(* CODESYS project 1_2_3_plc_chalet_xplanar.library
   Title: CHALET_XPlanar
   Version: 1.2.3
   Placeholder: CHALET_XPlanar
   Company: Beckhoff CH

Project tree, tasks and I/O mapping:
  libraries: CHALET_BaseComponents, * (Beckhoff CH); Tc2_Math, * (Beckhoff Automation GmbH); Tc2_Standard, 3.3.3.0 (Beckhoff Automation GmbH); Tc2_System, 3.4.25.0 (Beckhoff Automation GmbH); Tc2_Utilities, 3.3.52.0 (Beckhoff Automation GmbH); Tc3_EventLogger, 3.1.30.0 (Beckhoff Automation GmbH); Tc3_JsonXml, 3.3.18.0 (Beckhoff Automation GmbH); Tc3_Mc3PlanarMotion, 3.1.10.11 (Beckhoff Automation GmbH); Tc3_Module, 3.3.21.0 (Beckhoff Automation GmbH); Tc3_Physics, 3.1.10.3 (Beckhoff Automation GmbH); Tc3_XPlanarUtility, 3.1.2203.3 (Beckhoff Automation GmbH & Co. KG)
  COMPONENTs/
    Casting/
      function ToMover [ST]
      function ToMoverPair [ST]
      function ToStation [ST]
      function ToTrack [ST]
    Environment/
      CD_XP_Environment
      function block FB_XP_Environment [ST]: AddToGroup, RemoveFromGroup, Clear, Configure, FB_init, HR, Initialize, OID, PlanarEnvironment, Update, UtilityEnvirement
      interface I_XP_Environment: AddToGroup, Clear, Configure, HR, Initialize, OID, PlanarEnvironment, RemoveFromGroup, Update, UtilityEnvirement
    Group/
      CD_XP_Groups
      function block FB_XP_Group [ST]: AddEnvironment, AddMover, AddTrack, Disable, Enable, FB_init, HR, Initialize, OID, Reset, Update
      interface I_XP_Group: AddEnvironment, AddMover, AddTrack, Disable, Enable, HR, Initialize, OID, Reset, Update
    Mover/
      Pair/
        function block FB_XP_MoverPair [ST]: FB_init, MoverMaster, MoverSlave
        interface I_XP_MoverPair: MoverMaster, MoverSlave
      Single/
        function block FB_XP_Mover [ST]: AddToGroup, RemoveFromGroup, MoveC, Disable, Enable, Reset, JoinTrack, MoveOnTrack, PositionOnTrack, CurrentStation, DistToTrack, FB_init, Halt, HR, Initialize, Mode, OID, PlanarMover, TargetStation, TcIoXPlanarMover, Update, UpdatePosition, UtilityMover
        interface I_XP_Mover: AddToGroup, RemoveFromGroup, MoveC, Disable, Enable, Reset, JoinTrack, MoveOnTrack, PositionOnTrack, CurrentStation, DistToTrack, Halt, HR, Mode, OID, PlanarMover, TargetStation, TcIoXPlanarMover
        interface I_XP_Mover_PLC: OID, PlanarMover, TcIoXPlanarMover, UtilityMover
      CD_XP_Movers
    Stationen/
      function block FB_XP_Station_Base [ST]: Configure, Configuring, PlcIfaceToMover, AccocietedTrack, AddMoverToQueue, AssignedMovers, CtsFreeMoverBuffer, DeleteMoversQueue, Feedback, InterfaceToMover, IsMoverInStation, PositionOnTrack, PositionXY, Ready, SearchPathToTarged, SendMoverToGroup, SendMoverToGroupExp, StationGroupID, Update
      function block FB_XP_Station_FBinit [ST]: Configuring, FB_init
      function block FB_XP_Station_JSON [ST]: Configuring, FB_init
      interface I_XP_Station: AccocietedTrack, AddMoverToQueue, AssignedMovers, Configure, Configuring, DeleteMoversQueue, PositionOnTrack, SearchPathToTarged, SendMoverToGroup, SendMoverToGroupExp, StationGroupID, Update
      interface I_XP_Station_PLC: AccocietedTrack, Feedback, IsMoverInStation, PlcIfaceToMover, PositionOnTrack, PositionXY, Ready, SendMoverToGroup, StationGroupID
      Klassendiagramm
      data type ST_PathFinder
    System/
      CD_XP_System
      CD_XP_System_Objects
      function block FB_XP_System [ST]: Disable, Disabled, Disabling, Enable, Enabled, Enabling, Station, ValidLUID, LinkEnvironment, LinkGroup, RegisterMover, RegisterMoverPair, RegisterStation, RegisterTrack, JoiningStation, JoiningTrack, Enviroment, Feedback, Initialize, Movers, Stations, Tracks, Update
      interface I_XP_System_PLC: Disable, Disabled, Enable, Enabled, Feedback, Initialize, Station, Update, ValidLUID
      interface I_XP_System_Registration: Enviroment, LinkEnvironment, LinkGroup, Movers, RegisterMover, RegisterMoverPair, RegisterStation, RegisterTrack, Stations, Tracks
    Track/
      CD_XP_Track
      function block FB_XP_Track_Base [ST]: AddToGroup, RemoveFromGroup, AddMover, CalcTrackPoints, Configure, Configuring, Disable, Enable, FB_init, HR, Length, OID, PlanarTrack, Reset, Update
      function block FB_XP_Track_JSON [ST]: ReadCenter, ReadDirection, ReadEnd, ReadStart, Configuring
      function block FB_XP_Track_TcCom [ST]: Configuring
      interface I_XP_Track: AddMover, AddToGroup, CalcTrackPoints, Configure, Configuring, Disable, Enable, HR, Length, OID, PlanarTrack, RemoveFromGroup, Reset
    Class Diagram_Iface
  00000000-0000-0000-0000-000000000000|Disclaimer Standard DE R1006.pdf
  Disclaimer Standard DE R1006.pdf
  global variables XPlanarParameterlist
*)

// COMPONENTs/Stationen/ST_PathFinder
TYPE ST_PathFinder :
STRUCT
	bTargetFound : BOOL; // Targed Station found on this path. No information about ready or not	
	nDistToTarget : INT;
	iFoundStation : I_CH_Object;
END_STRUCT
END_TYPE

// XPlanarParameterlist
{attribute 'qualified_only'}
VAR_GLOBAL CONSTANT 
	(*Minimum gap center to center on track *)
	F_MOVER_MINIMUM_GAP_ON_TRACK : LREAL := 200.0;

	(*Additional gap center to center on track *)
	F_MOVER_ADDITIONAL_GAP_ON_TRACK : LREAL := 60.0;
	
	(*Pathfinder max recursion search depth in stations*)
	N_MAX_SEARCH_DEPTH: INT := 5;
		
	(*Use the automatic deployment function to copy the .JSON files to the %TC_BOOTPRJPATH%OCFG at Activate configuration*)
	S_JSON_FOLDER_PATH_ON_TARGED : STRING := 'C:\TwinCAT\3.1\Boot\OCFG\';
	
	(*get an array of points of track in this size *)
	N_TRACE_POINTS : UINT := 30;
END_VAR

// COMPONENTs/Casting/ToMover
FUNCTION ToMover : BOOL
VAR_INPUT
	iChObject : I_CH_OBJECT;
	iXpMover : Reference to I_XP_Mover;
END_VAR

VAR
	iTmp : I_XP_Mover;
END_VAR

(* 
   1. Test if the interface exists
   2. Test if the object implements a "Object" interface 
   3. Write reference to interface in parameter
   4. Returne TRUE if succesfull
*)
IF iChObject <> 0 AND_THEN __QUERYINTERFACE(iChObject,iTmp) THEN
	iXpMover := iTmp;
	ToMover := TRUE;
END_IF

END_FUNCTION

// COMPONENTs/Mover/Single/I_XP_Mover
INTERFACE I_XP_Mover EXTENDS __SYSTEM.IQueryInterface

METHOD AddToGroup : HRESULT
VAR_INPUT
	iGroup : I_XP_Group;
END_VAR
END_METHOD

METHOD RemoveFromGroup : HRESULT
END_METHOD

METHOD MoveC : HRESULT
VAR_INPUT
	fPosition : LREAL;
END_VAR
END_METHOD

METHOD Disable : HRESULT
VAR_INPUT
END_VAR
END_METHOD

METHOD Enable : HRESULT
VAR_INPUT
END_VAR
END_METHOD

METHOD Reset : HRESULT
VAR_INPUT
END_VAR
END_METHOD

METHOD JoinTrack : HRESULT
VAR_INPUT
	iTrack : I_XP_Track;
END_VAR
END_METHOD

METHOD MoveOnTrack : HRESULT
VAR_INPUT
	iTrack : I_XP_Track;
	fPosition : LREAL;
END_VAR
END_METHOD

PROPERTY PositionOnTrack : Lreal
GET
END_GET
END_PROPERTY

{attribute 'monitoring':='call'}
PROPERTY CurrentStation : STRING
GET
END_GET
SET
END_SET
END_PROPERTY

METHOD DistToTrack : LREAL
VAR_INPUT
	iTrack : I_XP_Track;
END_VAR
END_METHOD

METHOD Halt : HRESULT
VAR_INPUT
END_VAR
END_METHOD

{attribute 'monitoring':='call'}
PROPERTY HR : HRESULT
GET
END_GET
END_PROPERTY

{attribute 'monitoring':='call'}
PROPERTY Mode : MC_PLANAR_MOVER_COMMAND_MODE
GET
END_GET
END_PROPERTY

{attribute 'monitoring':='call'}
PROPERTY OID : OTCID
GET
END_GET
END_PROPERTY

{attribute 'monitoring':='call'}
PROPERTY PlanarMover : REFERENCE TO MC_PlanarMover
GET
END_GET
END_PROPERTY

{attribute 'monitoring':='call'}
PROPERTY TargetStation : String
GET
END_GET
SET
END_SET
END_PROPERTY

PROPERTY TcIoXPlanarMover : Tc3_XPlanarUtility.I_TcIoXPlanarMover
GET
END_GET
END_PROPERTY

END_INTERFACE

// COMPONENTs/Group/I_XP_Group
INTERFACE I_XP_Group

METHOD AddEnvironment : HRESULT
VAR_INPUT
	refEnvironment : REFERENCE TO MC_PlanarEnvironment;
	refFeedback : REFERENCE TO MC_PlanarFeedback;
END_VAR
END_METHOD

METHOD AddMover : HRESULT
VAR_INPUT
	refMover : REFERENCE TO MC_PlanarMover;
	refFeedback : REFERENCE TO MC_PlanarFeedback;
END_VAR
END_METHOD

METHOD AddTrack : HRESULT
VAR_INPUT
	refTrack : REFERENCE TO MC_PlanarTrack;
	refFeedback : REFERENCE TO MC_PlanarFeedback;
END_VAR
END_METHOD

METHOD Disable : HRESULT
VAR_INPUT
END_VAR
END_METHOD

METHOD Enable : HRESULT
VAR_INPUT
END_VAR
END_METHOD

{attribute 'monitoring':='call'}
PROPERTY HR : HRESULT
GET
END_GET
END_PROPERTY

METHOD Initialize : HRESULT
VAR_INPUT
END_VAR
END_METHOD

{attribute 'monitoring':='call'}
PROPERTY OID : OTCID
GET
END_GET
END_PROPERTY

METHOD Reset : HRESULT
VAR_INPUT
END_VAR
END_METHOD

METHOD PUBLIC Update : HRESULT
VAR_INPUT
END_VAR
END_METHOD

END_INTERFACE

// COMPONENTs/Track/I_XP_Track
INTERFACE I_XP_Track

METHOD AddMover : HRESULT
VAR_INPUT
	refMover : REFERENCE TO MC_PlanarMover;
	refFeedback : REFERENCE TO MC_PlanarFeedback;
END_VAR
END_METHOD

METHOD AddToGroup : HRESULT
VAR_INPUT
	iGroup : I_XP_Group;
END_VAR
END_METHOD

METHOD CalcTrackPoints : HRESULT
VAR_INPUT
END_VAR
END_METHOD

METHOD Configure : HRESULT
VAR_INPUT
END_VAR
END_METHOD

METHOD Configuring : HRESULT
VAR_INPUT
END_VAR
END_METHOD

METHOD Disable : HRESULT
VAR_INPUT
END_VAR
END_METHOD

METHOD Enable : HRESULT
VAR_INPUT
END_VAR
END_METHOD

{attribute 'monitoring':='call'}
PROPERTY HR : HRESULT
GET
END_GET
END_PROPERTY

{attribute 'monitoring':='call'}
PROPERTY Length : LREAL
GET
END_GET
END_PROPERTY

{attribute 'monitoring':='call'}
PROPERTY OID : OTCID
GET
END_GET
END_PROPERTY

{attribute 'monitoring':='call'}
PROPERTY PlanarTrack : REFERENCE TO MC_PlanarTrack
GET
END_GET
END_PROPERTY

METHOD RemoveFromGroup : HRESULT
END_METHOD

METHOD Reset : HRESULT
VAR_INPUT
END_VAR
END_METHOD

END_INTERFACE

// COMPONENTs/Casting/ToMoverPair
FUNCTION ToMoverPair : BOOL
VAR_INPUT
	iChObject : I_CH_OBJECT;
	iXpMoverPair : Reference to I_XP_MoverPair;
END_VAR

VAR
	iTmp : I_XP_MoverPair;
END_VAR

(* 
   1. Test if the interface exists
   2. Test if the object implements a "Object" interface 
   3. Write reference to interface in parameter
   4. Returne TRUE if succesfull
*)
IF iChObject <> 0 AND_THEN __QUERYINTERFACE(iChObject,iTmp) THEN
	iXpMoverPair := iTmp;
	ToMoverPair := TRUE;
END_IF

END_FUNCTION

// COMPONENTs/Mover/Pair/I_XP_MoverPair
INTERFACE I_XP_MoverPair

{attribute 'monitoring':='call'}
PROPERTY MoverMaster : I_XP_Mover
GET
END_GET
SET
END_SET
END_PROPERTY

{attribute 'monitoring':='call'}
PROPERTY MoverSlave : I_XP_Mover
GET
END_GET
SET
END_SET
END_PROPERTY

END_INTERFACE

// COMPONENTs/Casting/ToStation
FUNCTION ToStation : BOOL
VAR_INPUT
	iChObject : I_CH_OBJECT;
	iXpStation : REFERENCE TO I_XP_Station;
END_VAR

VAR
	iTmp : I_XP_Station;
END_VAR

(* Register the Station
   1. Test if the interface exists
   2. Test if the object implements a "Object" interface 
*)
IF iChObject <> 0 AND_THEN __QUERYINTERFACE(iChObject,iTmp) THEN
	iXpStation := iTmp;
	ToStation := TRUE;
END_IF

END_FUNCTION

// COMPONENTs/Stationen/I_XP_Station
INTERFACE I_XP_Station EXTENDS __SYSTEM.IQueryInterface

{attribute 'monitoring':='call'}
PROPERTY AccocietedTrack : I_XP_Track
GET
END_GET
END_PROPERTY

METHOD AddMoverToQueue : HRESULT
VAR_INPUT
	iMover : I_CH_Object;
END_VAR
END_METHOD

PROPERTY AssignedMovers : I_CH_List
GET
END_GET
END_PROPERTY

METHOD Configure : HRESULT
END_METHOD

METHOD Configuring : HRESULT
END_METHOD

METHOD DeleteMoversQueue : HRESULT
VAR_INPUT
END_VAR
END_METHOD

PROPERTY PositionOnTrack : LREAL
GET
END_GET
END_PROPERTY

METHOD SearchPathToTarged : ST_PathFinder
VAR_INPUT
	sTargedStationGroupId	: STRING;
	nSearchDepth		: INT;
END_VAR
END_METHOD

METHOD SendMoverToGroup : I_CH_Feedback
VAR_INPUT 
	sTargedStationGroupID : STRING;
END_VAR
END_METHOD

METHOD SendMoverToGroupExp : HRESULT
VAR_INPUT
	sTargedStationGroupID : STRING;
	iMover : I_XP_Mover;
END_VAR
END_METHOD

{attribute 'monitoring':='call'}
PROPERTY StationGroupID : STRING
GET
END_GET
END_PROPERTY

METHOD Update : HRESULT
VAR_INPUT
END_VAR
END_METHOD

END_INTERFACE

// COMPONENTs/Casting/ToTrack
FUNCTION ToTrack : BOOL
VAR_INPUT
	iChObject : I_CH_OBJECT;
	iXpTrack : REFERENCE TO I_XP_Track;
END_VAR

VAR
	iTmp : I_XP_Track;
END_VAR

(* 
   1. Test if the interface exists
   2. Test if the object implements a "Object" interface 
   3. Write reference to interface in parameter
   4. Returne TRUE if succesfull
*)
IF iChObject <> 0 AND_THEN __QUERYINTERFACE(iChObject,iTmp) THEN
	iXpTrack := iTmp;
	ToTrack := TRUE;
END_IF

END_FUNCTION

// COMPONENTs/Environment/FB_XP_Environment
{attribute 'no_explicit_call' := '[FB_ImageSource] Do not call the body - Stick to OOP'}
FUNCTION_BLOCK FB_XP_Environment EXTENDS FB_CH_Object IMPLEMENTS I_XP_Environment
VAR
	fbEnvironment : MC_PlanarEnvironment;
	fbUtilityEnvirement : FB_TcIoXPlanarEnvironment;
	{attribute 'hide'}
	iXpSystem : I_XP_System_Registration;
	fbActiveCmd : MC_PlanarFeedback;

END_VAR

METHOD AddToGroup : HRESULT
VAR_INPUT
	iGroup : I_XP_Group;
END_VAR
IF NOT THIS^.fbActiveCmd.Busy AND NOT THIS^.fbActiveCmd.Busy THEN
	iGroup.AddEnvironment(THIS^.fbEnvironment, THIS^.fbActiveCmd);
	AddToGroup := S_OK;
ELSE
	AddToGroup := S_FALSE;
END_IF
END_METHOD

METHOD RemoveFromGroup : HRESULT
IF NOT THIS^.fbActiveCmd.Busy THEN
	THIS^.fbEnvironment.RemoveFromGroup(THIS^.fbActiveCmd);
	RemoveFromGroup := S_OK;
ELSE
	RemoveFromGroup := S_FALSE;
END_IF
END_METHOD

METHOD Clear : HRESULT
THIS^.fbEnvironment.Clear(commandFeedback:=THIS^.fbActiveCmd);
Clear := S_OK;
END_METHOD

METHOD Configure : HRESULT
// To be automatically read from the Utility Stator info
// 06.2022 is read automaticli if Envirement Init Parameter has a link to XPLANAR TcCom Object.

THIS^.fbEnvironment.CreateBoundary(commandFeedback:=THIS^.fbActiveCmd);
Configure := S_OK;
END_METHOD

METHOD FB_init : BOOL
VAR_INPUT
	bInitRetains : BOOL; // if TRUE, the retain variables are initialized (warm start / cold start)
	bInCopyCode : BOOL;  // if TRUE, the instance afterwards gets moved into the copy code (online change)
	oSystem : I_CH_Object;
END_VAR
(* Register to the Xplanar System
   1. Test if the interface exists
   2. Test if the object implements a "System for Mover" interface 
*)
IF oSystem <> 0 AND_THEN __QUERYINTERFACE(oSystem,THIS^.iXpSystem) THEN
	THIS^.iXpSystem.LinkEnvironment(THIS^);
END_IF
END_METHOD

{attribute 'monitoring':='call'}
PROPERTY HR : HRESULT
GET
IF THIS^.fbActiveCmd.Busy THEN
	HR := S_PENDING;
END_IF

IF THIS^.fbActiveCmd.Done THEN
	HR := S_OK;
END_IF

IF THIS^.fbActiveCmd.Error THEN
	HR := E_FAIL;
END_IF
END_GET
END_PROPERTY

METHOD Initialize : HRESULT
VAR_INST
	bInitDone :BOOL := FALSE;
END_VAR
IF NOT bInitDone THEN
	Initialize := S_PENDING;
	IF fbUtilityEnvirement.Init(bExecute := TRUE) THEN
		fbUtilityEnvirement.Init(bExecute := FALSE);
		bInitDone := TRUE;
	END_IF
ELSE	
	Initialize := S_OK;
END_IF
END_METHOD

{attribute 'monitoring':='call'}
PROPERTY OID : OTCID
GET
OID := THIS^.fbEnvironment.MCTOPLC_STD.EnvironmentOID;
END_GET
END_PROPERTY

{attribute 'monitoring':='call'}
PROPERTY PlanarEnvironment : REFERENCE TO MC_PlanarEnvironment
GET
PlanarEnvironment ref= THIS^.fbEnvironment;
END_GET
END_PROPERTY

METHOD PUBLIC Update : HRESULT
VAR_INPUT
END_VAR
THIS^.fbEnvironment.Update();
fbActiveCmd.Update();
END_METHOD

PROPERTY UtilityEnvirement : Tc3_XPlanarUtility.I_Environment
GET
UtilityEnvirement := fbUtilityEnvirement;
END_GET
END_PROPERTY

END_FUNCTION_BLOCK

// COMPONENTs/Environment/I_XP_Environment
INTERFACE I_XP_Environment

METHOD AddToGroup : HRESULT
VAR_INPUT
	iGroup : I_XP_Group;
END_VAR
END_METHOD

METHOD Clear : HRESULT
END_METHOD

METHOD Configure : HRESULT
VAR_INPUT
END_VAR
END_METHOD

{attribute 'monitoring':='call'}
PROPERTY HR : HRESULT
GET
END_GET
END_PROPERTY

METHOD Initialize : HRESULT
END_METHOD

{attribute 'monitoring':='call'}
PROPERTY OID : OTCID
GET
END_GET
END_PROPERTY

{attribute 'monitoring':='call'}
PROPERTY PlanarEnvironment : REFERENCE TO MC_PlanarEnvironment
GET
END_GET
END_PROPERTY

METHOD RemoveFromGroup : HRESULT
END_METHOD

METHOD PUBLIC Update : HRESULT
VAR_INPUT
END_VAR
END_METHOD

PROPERTY UtilityEnvirement : Tc3_XPlanarUtility.I_Environment
GET
END_GET
END_PROPERTY

END_INTERFACE

// COMPONENTs/System/I_XP_System_Registration
INTERFACE I_XP_System_Registration

PROPERTY Enviroment : I_XP_Environment
GET
END_GET
END_PROPERTY

METHOD LinkEnvironment : HRESULT
VAR_INPUT
	oEnvironment : I_CH_Object;
END_VAR
END_METHOD

METHOD LinkGroup : HRESULT
VAR_INPUT
	oGroup : I_CH_Object;
END_VAR
END_METHOD

PROPERTY Movers : I_CH_LIST
GET
END_GET
END_PROPERTY

METHOD RegisterMover : HRESULT
VAR_INPUT
	oMover : I_CH_Object;
END_VAR
END_METHOD

METHOD RegisterMoverPair : HRESULT
VAR_INPUT
	oMoverPair : I_CH_Object;
END_VAR
END_METHOD

METHOD RegisterStation : HRESULT
VAR_INPUT
	oStation : I_CH_Object;
END_VAR
END_METHOD

METHOD RegisterTrack : HRESULT
VAR_INPUT
	oTrack : I_CH_Object;
END_VAR
END_METHOD

PROPERTY Stations : I_CH_LIST
GET
END_GET
END_PROPERTY

PROPERTY Tracks : I_CH_LIST
GET
END_GET
END_PROPERTY

END_INTERFACE

// COMPONENTs/Group/FB_XP_Group
{attribute 'no_explicit_call' := '[FB_ImageSource] Do not call the body - Stick to OOP'}
FUNCTION_BLOCK FB_XP_Group EXTENDS FB_CH_Object IMPLEMENTS I_XP_Group
VAR
	fbGroup : MC_PlanarGroup;
	{attribute 'hide'}
	iXpSystem : I_XP_System_Registration;
	fbActiveCmd : MC_PlanarFeedback;
END_VAR

METHOD AddEnvironment : HRESULT
VAR_INPUT
	refEnvironment : REFERENCE TO MC_PlanarEnvironment;
	refFeedback : REFERENCE TO MC_PlanarFeedback;
END_VAR
refEnvironment.AddToGroup(refFeedback, fbGroup);
END_METHOD

METHOD AddMover : HRESULT
VAR_INPUT
	refMover : REFERENCE TO MC_PlanarMover;
	refFeedback : REFERENCE TO MC_PlanarFeedback;
END_VAR
refMover.AddToGroup(refFeedback, fbGroup);
END_METHOD

METHOD AddTrack : HRESULT
VAR_INPUT
	refTrack : REFERENCE TO MC_PlanarTrack;
	refFeedback : REFERENCE TO MC_PlanarFeedback;
END_VAR
refTrack.AddToGroup(refFeedback, fbGroup);
END_METHOD

METHOD Disable : HRESULT
VAR_INPUT
END_VAR
IF NOT THIS^.fbActiveCmd.Busy THEN
	THIS^.fbGroup.Disable(fbActiveCmd);
	Disable := S_OK;
ELSE
	Disable := S_FALSE;
END_IF
END_METHOD

METHOD Enable : HRESULT
VAR_INPUT
END_VAR
IF NOT THIS^.fbActiveCmd.Busy THEN
	THIS^.fbGroup.Enable(fbActiveCmd);
	Enable := S_OK;
ELSE
	Enable := S_FALSE;
END_IF
END_METHOD

METHOD FB_init : BOOL
VAR_INPUT
	bInitRetains : BOOL; // if TRUE, the retain variables are initialized (warm start / cold start)
	bInCopyCode : BOOL;  // if TRUE, the instance afterwards gets moved into the copy code (online change)
	oSystem : I_CH_Object;
END_VAR
(* Register to the Xplanar System
   1. Test if the interface exists
   2. Test if the object implements a "System for Mover" interface 
*)
IF oSystem <> 0 AND_THEN __QUERYINTERFACE(oSystem,THIS^.iXpSystem) THEN
	THIS^.iXpSystem.LinkGroup(THIS^);
END_IF
END_METHOD

{attribute 'monitoring':='call'}
PROPERTY HR : HRESULT
GET
IF THIS^.fbActiveCmd.Busy THEN
	HR := S_PENDING;
END_IF

IF THIS^.fbActiveCmd.Done THEN
	HR := S_OK;
END_IF

IF THIS^.fbActiveCmd.Error THEN
	HR := E_FAIL;
END_IF
END_GET
END_PROPERTY

METHOD Initialize : HRESULT
VAR_INPUT
END_VAR
Initialize := S_OK;
END_METHOD

{attribute 'monitoring':='call'}
PROPERTY OID : OTCID
GET
OID := THIS^.fbGroup.MCTOPLC_STD.GroupOID;
END_GET
END_PROPERTY

METHOD Reset : HRESULT
VAR_INPUT
END_VAR
IF NOT THIS^.fbActiveCmd.Busy THEN
	THIS^.fbGroup.Reset(fbActiveCmd);
	Reset := S_OK;
ELSE
	Reset := S_FALSE;
END_IF
END_METHOD

METHOD PUBLIC Update : HRESULT
VAR_INPUT
END_VAR
THIS^.fbGroup.Update();
fbActiveCmd.Update();
END_METHOD

END_FUNCTION_BLOCK

// COMPONENTs/Mover/Pair/FB_XP_MoverPair
FUNCTION_BLOCK FB_XP_MoverPair EXTENDS FB_CH_Object IMPLEMENTS I_XP_MoverPair
VAR
	{attribute 'hide'}
    iMoverMaster : I_XP_Mover;
	{attribute 'hide'}
    iMoverSlave  : I_XP_Mover;
	{attribute 'hide'}
    iXpSystem    : I_XP_System_Registration;
END_VAR

METHOD FB_init : BOOL
VAR_INPUT
	bInitRetains : BOOL; // if TRUE, the retain variables are initialized (warm start / cold start)
	bInCopyCode : BOOL;  // if TRUE, the instance afterwards gets moved into the copy code (online change)
	oSystem : I_CH_Object;
END_VAR

VAR
	iXpSystem : I_XP_System_Registration;
END_VAR
(* Register to the Xplanar System
   1. Test if the interface exists
   2. Test if the object implements a "System for Mover" interface 
*)
IF oSystem <> 0 AND_THEN __QUERYINTERFACE(oSystem,THIS^.iXpSystem) THEN
	THIS^.iXpSystem.RegisterMoverPair(THIS^);
END_IF
END_METHOD

{attribute 'monitoring':='call'}
PROPERTY MoverMaster : I_XP_Mover
GET
MoverMaster := THIS^.iMoverMaster;
END_GET
SET
THIS^.iMoverMaster := MoverMaster;
END_SET
END_PROPERTY

{attribute 'monitoring':='call'}
PROPERTY MoverSlave : I_XP_Mover
GET
MoverSlave := THIS^.iMoverSlave;
END_GET
SET
THIS^.iMoverSlave := MoverSlave;
END_SET
END_PROPERTY

END_FUNCTION_BLOCK

// COMPONENTs/Mover/Single/FB_XP_Mover
// The warning " Interface of overridden methode xxx of base I_xxx doesn't match declaration" can be disabled here. 
{warning disable C0094 }

FUNCTION_BLOCK FB_XP_Mover EXTENDS FB_CH_Object IMPLEMENTS I_XP_Mover, I_XP_Mover_PLC
VAR
	fbMover : MC_PlanarMover;
	fbActiveCmd : MC_PlanarFeedback;	
	
	{attribute 'hide'} 
	fbUtilityMover : FB_McPlanarMover;
	{attribute 'hide'}
	iXpSystem : I_XP_System_Registration;
	{attribute 'hide'} 
	stPosition : PositionXYC;
	{attribute 'hide'} 
	sTargedStation : STRING;
	{attribute 'hide'} 
	sCurrentStation : STRING;
END_VAR

{warning restore C0094}

METHOD AddToGroup : HRESULT
VAR_INPUT
	iGroup : I_XP_Group;
END_VAR
IF NOT THIS^.fbActiveCmd.Busy THEN
	iGroup.AddMover(THIS^.fbMover, THIS^.fbActiveCmd);
	AddToGroup := S_OK;
ELSE
	AddToGroup := S_FALSE;
END_IF
END_METHOD

METHOD RemoveFromGroup : HRESULT

VAR
	iGroup: INT;
END_VAR
IF NOT THIS^.fbActiveCmd.Busy THEN
	THIS^.fbMover.RemoveFromGroup(THIS^.fbActiveCmd);
	RemoveFromGroup := S_OK;
ELSE
	RemoveFromGroup := S_FALSE;
END_IF
END_METHOD

METHOD MoveC : HRESULT
VAR_INPUT
	fPosition : LREAL;
END_VAR

THIS^.fbMover.MoveC(commandFeedback	:= THIS^.fbActiveCmd, 
					targetPosition	:= fPosition, 
					constraint		:= 0, 
					options			:= 0
					);

MoveC := S_OK;
END_METHOD

METHOD Disable : HRESULT
VAR_INPUT
END_VAR
THIS^.fbMover.Disable(THIS^.fbActiveCmd);
Disable := S_OK;
END_METHOD

METHOD Enable : HRESULT
VAR_INPUT
END_VAR
IF NOT THIS^.fbActiveCmd.Busy THEN
	THIS^.fbMover.Enable(fbActiveCmd);
	Enable := S_OK;
ELSE
	Enable := S_FALSE;
END_IF
END_METHOD

METHOD Reset : HRESULT
VAR_INPUT
END_VAR
THIS^.fbMover.Reset(THIS^.fbActiveCmd);
Reset := S_OK;
END_METHOD

METHOD JoinTrack : HRESULT
VAR_INPUT
	iTrack : I_XP_Track;
END_VAR

VAR
	//iTrack : I_XP_Track;
END_VAR
IF NOT THIS^.fbActiveCmd.Busy THEN
	iTrack.AddMover(THIS^.fbMover, THIS^.fbActiveCmd);
	JoinTrack := S_OK;
ELSE
	JoinTrack := S_FALSE;
END_IF
END_METHOD

METHOD MoveOnTrack : HRESULT
VAR_INPUT
	iTrack : I_XP_Track;
	fPosition : LREAL;
END_VAR

VAR
	moveOptions: ST_MoveOnTrackOptions;
	fMoverDiagonal : LREAL;
END_VAR
moveOptions.direction := MC_DIRECTION.mcDirectionPositive;
moveOptions.additionalTurns := 0;

//gap = Pythagoras diagonal + x mm, minimum x mm
fMoverDiagonal := SQRT(EXPT((THIS^.fbUtilityMover.GetMoverHeight()),2)+EXPT((THIS^.fbUtilityMover.GetMoverWidth()),2));
moveOptions.gap := MAX(XPlanarParameterlist.F_MOVER_MINIMUM_GAP_ON_TRACK ,fMoverDiagonal + XPlanarParameterlist.F_MOVER_ADDITIONAL_GAP_ON_TRACK );

IF iTrack <> 0 THEN
	THIS^.fbMover.MoveOnTrack(
		commandFeedback:=THIS^.fbActiveCmd,
		targetTrack:=iTrack.PlanarTrack, 
		targetPositionOnTrack:=fPosition, 
		constraint:=0, 
		options:=moveOptions);
	MoveOnTrack := S_OK;
ELSE
	MoveOnTrack := S_FALSE;
END_IF
END_METHOD

PROPERTY PositionOnTrack : LREAL
GET
VAR
	fbMoverSetPosOnTrack: Tc3_XPlanarUtility.ST_MCMoverSetPosOnTrack;
END_VAR
fbMoverSetPosOnTrack := THIS^.fbUtilityMover.GetPositionOnTrack();
PositionOnTrack := fbMoverSetPosOnTrack.SetPos;
END_GET
END_PROPERTY

{attribute 'monitoring':='call'}
PROPERTY CurrentStation : STRING
GET
CurrentStation := THIS^.sCurrentStation;
END_GET
SET
THIS^.sCurrentStation := currentStation;
END_SET
END_PROPERTY

METHOD DistToTrack : LREAL
VAR_INPUT
	iTrack : I_XP_Track;
END_VAR
VAR
	fPositionOnTrack : LREAL;
	trackPosition : PositionXYC;
END_VAR
//get Pos on track in mm
fPositionOnTrack := iTrack.PlanarTrack.GetArcLengthClosestTo(geometry:=THIS^.stPosition);

//convert pos on track in XY
iTrack.PlanarTrack.GetPositionAt(arcLength := fPositionOnTrack, position:=trackPosition);

//get distance to mover
DistToTrack := SQRT(EXPT((trackPosition.x - THIS^.stPosition.x),2)+EXPT((trackPosition.y - THIS^.stPosition.y),2));
END_METHOD

METHOD FB_init : BOOL
VAR_INPUT
	bInitRetains : BOOL; // if TRUE, the retain variables are initialized (warm start / cold start)
	bInCopyCode : BOOL;  // if TRUE, the instance afterwards gets moved into the copy code (online change)
	oSystem : I_CH_Object;
END_VAR
(* Register to the Xplanar System
   1. Test if the interface exists
   2. Test if the object implements a "System for Mover" interface 
*)
IF oSystem <> 0 AND_THEN __QUERYINTERFACE(oSystem,THIS^.iXpSystem) THEN
	THIS^.iXpSystem.RegisterMover(THIS^);
END_IF
END_METHOD

METHOD Halt : HRESULT
VAR_INPUT
END_VAR
THIS^.fbMover.Halt(THIS^.fbActiveCmd,0);

Halt := S_OK;
END_METHOD

{attribute 'monitoring':='call'}
PROPERTY HR : HRESULT
GET
IF THIS^.fbActiveCmd.Busy THEN 
	HR := S_PENDING;
END_IF

IF THIS^.fbActiveCmd.Done THEN 
	HR := S_OK;
END_IF

IF THIS^.fbActiveCmd.Error THEN 
	HR := E_FAIL;
END_IF
END_GET
END_PROPERTY

METHOD Initialize : HRESULT
VAR_INST
	bInitDone :BOOL := FALSE;
END_VAR
VAR
	//nLoopIndex : UINT;
	
	//zzzMover : I_TcIoXPlanarMover;
	//zzzTcIoXPlanar : I_TcIoXPlanarProcessingUnit;
	//zzzOid : OTCID;
	//zzzIENv : I_XP_Environment;
END_VAR
IF NOT bInitDone THEN
	Initialize := S_PENDING;
	
	//braucht es das noch? zzz
	//IF iXpSystem.Enviroment.Initialize() <> S_OK  THEN
	//	//wait until init of FB_TcIoXPlanarEnvironment is done.
	//	RETURN;
	//END_IF
	//
    //
	//IF fbUtilityMover.Init(bExecute:= TRUE, nObjectId:=THIS^.fbMover.MCTOPLC.STD.MoverOID) THEN
	//	fbUtilityMover.Init(bExecute:= FALSE, nObjectId:=THIS^.fbMover.MCTOPLC.STD.MoverOID);
	//ELSE
	//	RETURN;
	//END_IF
		
	bInitDone := TRUE;	
	
ELSE	
	Initialize := S_OK;	
END_IF
END_METHOD

{attribute 'monitoring':='call'}
PROPERTY Mode : MC_PLANAR_MOVER_COMMAND_MODE
GET
Mode := THIS^.fbMover.MCTOPLC.STD.CommandMode;
END_GET
END_PROPERTY

{attribute 'monitoring':='call'}
PROPERTY OID : OTCID
GET
OID := THIS^.fbMover.MCTOPLC.STD.MoverOID;
END_GET
END_PROPERTY

{attribute 'monitoring':='call'}
PROPERTY PlanarMover : REFERENCE TO MC_PlanarMover
GET
PlanarMover ref= THIS^.fbMover;
END_GET
END_PROPERTY

{attribute 'monitoring':='call'}
PROPERTY TargetStation : String
GET
TargetStation := THIS^.sTargedStation;
END_GET
SET
THIS^.sTargedStation := TargetStation;
END_SET
END_PROPERTY

{attribute 'monitoring':='call'}
PROPERTY TcIoXPlanarMover : Tc3_XPlanarUtility.I_TcIoXPlanarMover
GET
VAR
	nLoopIndex : UINT;
	zzzMover : I_TcIoXPlanarMover;
END_VAR
//TcIoXPlanarMover:= THIS^.iTcIoXPlanarMover;

FOR nLoopIndex := 1 TO UDINT_TO_UINT(Param_TcIoXPlanarEnvironment.MaxXPlanarMoversPerXpu) DO
	zzzMover := iXpSystem.Enviroment.UtilityEnvirement.XpuTcIo(1).MoverTcIo(nLoopIndex);
	IF zzzMover <> 0 AND_THEN zzzMover.GetNcMoverOid() = OID THEN
		TcIoXPlanarMover := iXpSystem.enviroment.UtilityEnvirement.XpuTcIo(1).MoverTcIo(nLoopIndex);
		RETURN;
	END_IF
END_FOR
END_GET
END_PROPERTY

METHOD PUBLIC Update : HRESULT
VAR_INPUT
END_VAR
THIS^.fbMover.Update();
THIS^.fbActiveCmd.Update();

THIS^.UpdatePosition();
END_METHOD

METHOD UpdatePosition : HRESULT
VAR_INPUT
END_VAR
THIS^.stPosition.x := THIS^.fbMover.MCTOPLC.ACT.ActPos.x;
THIS^.stPosition.y := THIS^.fbMover.MCTOPLC.ACT.ActPos.y;
THIS^.stPosition.c := THIS^.fbMover.MCTOPLC.ACT.ActPos.c;
END_METHOD

{attribute 'monitoring':='call'}
PROPERTY UtilityMover : I_McPlanarMover
GET
UtilityMover := THIS^.fbUtilityMover;
END_GET
END_PROPERTY

END_FUNCTION_BLOCK

// COMPONENTs/Mover/Single/I_XP_Mover_PLC
INTERFACE I_XP_Mover_PLC

{attribute 'monitoring':='call'}
PROPERTY OID : OTCID
GET
END_GET
END_PROPERTY

{attribute 'monitoring':='call'}
PROPERTY PlanarMover : REFERENCE TO MC_PlanarMover
GET
END_GET
END_PROPERTY

PROPERTY TcIoXPlanarMover : Tc3_XPlanarUtility.I_TcIoXPlanarMover
GET
END_GET
END_PROPERTY

{attribute 'monitoring':='call'}
PROPERTY UtilityMover : I_McPlanarMover
GET
END_GET
END_PROPERTY

END_INTERFACE

// COMPONENTs/Stationen/FB_XP_Station_Base
FUNCTION_BLOCK ABSTRACT FB_XP_Station_Base EXTENDS FB_CH_Object IMPLEMENTS I_XP_Station, I_XP_Station_PLC
VAR
	{attribute 'hide'}
	bReady 		: BOOL := TRUE;
	{attribute 'hide'}
	sStationGroupID : STRING;
	{attribute 'hide'}
	nCtsMinMovers : INT := 0;
	{attribute 'hide'}
	nCtsMaxMovers : INT := 1;
	{attribute 'hide'}	
	fbPosition : PositionXY;
	{attribute 'hide'}	
	fbJsonParser : FB_JsonDomParser;
	{attribute 'hide'}	
	nState_Configuring: INT;
	{attribute 'hide'}	
	iAccocietedTrack : I_XP_Track;
	{attribute 'hide'}	
	iXpSystem : I_XP_System_Registration;
	
	{attribute 'hide'}
	fbFeedback : FB_CH_Feedback;
	
	(*List of stations*)
	{attribute 'hide'}	
	fbStationsAhead : FB_CH_List;
	
	(* Lists to handle the ownership of movers *)
	{attribute 'hide'}
	fbAssignedMovers 			: FB_CH_List;		// Movers approaching the station

END_VAR

METHOD Configure : HRESULT
VAR_INPUT
END_VAR
THIS^.nState_Configuring := 10;

Configure := S_OK;
END_METHOD

METHOD Abstract Configuring : HRESULT
VAR_INPUT
END_VAR
END_METHOD

{attribute 'monitoring':='call'}
(* Return interface to mover in station. Return 0 if no mover is in station *)
PROPERTY PlcIfaceToMover : I_XP_Mover_PLC
GET
VAR
	iMover : I_XP_Mover;
END_VAR
iMover := THIS^.InterfaceToMover;

IF 	iMover <> 0 THEN
	__QUERYINTERFACE(iMover,PlcIfaceToMover);
END_IF
END_GET
END_PROPERTY

{attribute 'monitoring':='call'}
PROPERTY AccocietedTrack : I_XP_Track
GET
AccocietedTrack := THIS^.iAccocietedTrack;
END_GET
END_PROPERTY

METHOD AddMoverToQueue : HRESULT
VAR_INPUT
	iMover : I_CH_Object;
END_VAR
VAR 
	iXPMover : I_XP_Mover;
END_VAR
IF ToMover(iMover, iXpMover) THEN
	AddMoverToQueue := fbAssignedMovers.AddObject(iMover);
	iXpMover.CurrentStation := THIS^.sStationGroupID;
ELSE
	AddMoverToQueue := E_FAIL;
END_IF
END_METHOD

PROPERTY AssignedMovers : I_CH_List
GET
AssignedMovers := THIS^.fbAssignedMovers;
END_GET
END_PROPERTY

//Return the number of avaiable moverplaces in this station. Return -1 if Station is not ready
{attribute 'monitoring':='call'}
PROPERTY CtsFreeMoverBuffer : INT
GET
VAR
	nMoversTotal: UINT;
END_VAR
IF NOT bReady THEN
	CtsFreeMoverBuffer := -1;
	RETURN;
END_IF

nMoversTotal := THIS^.fbAssignedMovers.Size;
CtsFreeMoverBuffer := THIS^.nCtsMaxMovers - TO_INT(nMoversTotal);
END_GET
END_PROPERTY

METHOD DeleteMoversQueue : HRESULT
VAR_INPUT
END_VAR
fbAssignedMovers.Clear();

DeleteMoversQueue := S_OK;
END_METHOD

{attribute 'monitoring':='call'}
PROPERTY Feedback : I_CH_Feedback
GET
Feedback := THIS^.fbFeedback;
END_GET
END_PROPERTY

{attribute 'monitoring':='call'}
(* Return interface to mover in station. Return 0 if no mover is in station *)
PROPERTY InterfaceToMover : I_XP_Mover
GET
VAR
	oMover : I_CH_Object;
	iMover : I_XP_Mover;
END_VAR
VAR CONSTANT
	fToleranceMm : LREAL := 1.0; 
END_VAR
InterfaceToMover := 0;

//compare all movers in this station with the coordinats of the station
THIS^.fbAssignedMovers.ResetIterator();
WHILE THIS^.fbAssignedMovers.HasNextObject() DO
	oMover := THIS^.fbAssignedMovers.GetNextObject();
	IF ToMover(oMover,iMover) THEN
		IF iMover.TargetStation = THIS^.StationGroupID 
			AND (iMover.HR = S_OK) //No active move cmd= Pos reached
			//AND (ABS(iMover.PlanarMover.MCTOPLC.SET.SetPos.x -  THIS^.fbPosition.x)<=fToleranceMm) 
			//AND (ABS(iMover.PlanarMover.MCTOPLC.SET.SetPos.y -  THIS^.fbPosition.y)<=fToleranceMm) 
			THEN	
			InterfaceToMover := iMover;
			RETURN;
		END_IF
	END_IF
END_WHILE
END_GET
END_PROPERTY

//Return TRUE if an mover is exactly on the station coordinates and has this station as destination
{attribute 'monitoring':='call'}
PROPERTY IsMoverInStation : BOOL
GET
//If interface to first mover is valid
IsMoverInStation := THIS^.InterfaceToMover<>0;
END_GET
END_PROPERTY

PROPERTY PositionOnTrack : LREAL
GET
PositionOnTrack := THIS^.iAccocietedTrack.PlanarTrack.GetArcLengthClosestTo(geometry:= THIS^.fbPosition);
END_GET
END_PROPERTY

{attribute 'monitoring':='call'}
PROPERTY PositionXY : REFERENCE TO  PositionXY
GET
PositionXY REF= THIS^.fbPosition;
END_GET
END_PROPERTY

{attribute 'monitoring':='call'}
PROPERTY Ready : BOOL
GET
Ready := THIS^.bReady;
END_GET
SET
THIS^.bReady := Ready;
END_SET
END_PROPERTY

METHOD SearchPathToTarged : ST_PathFinder
VAR_INPUT
	sTargedStationGroupId	: STRING;
	nSearchDepth			: INT;
END_VAR

VAR
	iStation: I_XP_Station;
	tempPath : ST_PathFinder;
	bestPath : ST_PathFinder;
END_VAR
//This is the serched Station
IF THIS^.sStationGroupID = sTargedStationGroupId THEN
	searchPathToTarged.iFoundStation := (THIS^);
	searchPathToTarged.nDistToTarget := 0;
	searchPathToTarged.bTargetFound := TRUE;
	
	//Station is full/not ready and can not be used as next targed
	IF THIS^.CtsFreeMoverBuffer <= 0 THEN
		searchPathToTarged.iFoundStation := 0;
	END_IF
	RETURN;
END_IF	


//Abort
IF nSearchDepth = XPlanarParameterlist.N_MAX_SEARCH_DEPTH THEN
	searchPathToTarged.iFoundStation := 0;
	searchPathToTarged.nDistToTarget := 0;
	searchPathToTarged.bTargetFound := FALSE;
END_IF


//seach on all station ahead the shortest way to targed
bestPath.nDistToTarget := 32767;
THIS^.fbStationsAhead.ResetIterator();
WHILE THIS^.fbStationsAhead.HasNextObject() DO
	IF ToStation(THIS^.fbStationsAhead.GetNextObject(),iStation) THEN
		tempPath := iStation.searchPathToTarged(sTargedStationGroupId, nSearchDepth+1);
		tempPath.nDistToTarget := tempPath.nDistToTarget +1;		
		IF tempPath.bTargetFound AND ((tempPath.nDistToTarget <= bestPath.nDistToTarget AND tempPath.iFoundStation<>0) OR (tempPath.nDistToTarget <= bestPath.nDistToTarget AND bestPath.iFoundStation=0)) THEN
			bestPath := tempPath;
		END_IF
	END_IF
END_WHILE


//Only check if the station is empty to pass through, if the station is not where the mover starts(the mover is there at first position)
IF nSearchDepth <> 0 THEN
	//IF current station has object, its not posible to move direct to next station, in this case use this station as targed
	IF bestPath.bTargetFound AND (NOT THIS^.fbAssignedMovers.IsEmpty OR bestPath.iFoundStation = 0)THEN
		//If the currend station has some empty buffer, use this as targed, else clear target and try in station before again
		IF THIS^.CtsFreeMoverBuffer > 0 THEN
			bestPath.iFoundStation := (THIS^);
		ELSE
			bestPath.iFoundStation := 0; 
		END_IF
	END_IF
END_IF


searchPathToTarged := bestPath;
END_METHOD

METHOD SendMoverToGroup : I_CH_Feedback
VAR_INPUT 
	sTargedStationGroupID : STRING;
END_VAR
VAR
	iMover : I_XP_Mover;
	sCommand : STRING;
END_VAR
IF THIS^.fbFeedback.Error THEN
	//Error active/not ready
	THIS^.fbFeedback.LastCommandAccepted	:= FALSE;

ELSIF NOT THIS^.IsMoverInStation THEN
	//No Mover in Station
	THIS^.fbFeedback.LastCommandAccepted	:= FALSE;

ELSIF sTargedStationGroupID=''  THEN
	//No targed
	THIS^.fbFeedback.LastCommandAccepted	:= FALSE;
	
ELSE
	iMover := THIS^.InterfaceToMover;
	//search path and send away.
	THIS^.fbFeedback.HR := THIS^.sendMoverToGroupExp(sTargedStationGroupID:=sTargedStationGroupID, iMover);
	
	//build string with command
	sCommand := CONCAT(sCommand,'sendMover');
	sCommand := CONCAT(sCommand, UDINT_TO_STRING(iMover.OID));
	sCommand := CONCAT(sCommand,'ToGroup');
	sCommand := CONCAT(sCommand,sTargedStationGroupID);	
	
	//set fbFeedback
	THIS^.fbFeedback.ActiveCommand		 := sCommand;
	THIS^.fbFeedback.LastCommandAccepted := TRUE;
END_IF

sendMoverToGroup := THIS^.fbFeedback;
END_METHOD

METHOD SendMoverToGroupExp : HRESULT
VAR_INPUT
	sTargedStationGroupID : STRING;
	iMover : I_XP_Mover;
END_VAR

VAR
	iMoverObject : I_CH_Object;
	iStation: I_XP_Station;
	pathForMover: ST_PathFinder;
END_VAR
IF iMover <> 0 THEN
	
	//set targed
	iMover.TargetStation := sTargedStationGroupID;
	
	//get object
	iMoverObject := THIS^.iXpSystem.Movers.FindOID(iMover.OID);
	
	//init
	iStation := THIS^;
	
	//remove mover from station(the search path metohde maybe not found an solution if this station is already full.
	THIS^.fbAssignedMovers.RemoveObject(iMoverObject);
	
	//search best station
	pathForMover := THIS^.searchPathToTarged(sTargedStationGroupId:= iMover.TargetStation, nSearchDepth:=0);

	IF NOT pathForMover.bTargetFound THEN
		// no path found in maximum search depth - ERROR
		sendMoverToGroupExp := E_FAIL;
	ELSIF pathForMover.iFoundStation = 0 THEN
		// path found but no movement posible, next station is full
		sendMoverToGroupExp := S_FALSE;
	ELSIF ToStation(pathForMover.iFoundStation,iStation) THEN
		//path found. valide interface. move to station
		sendMoverToGroupExp := iMover.MoveOnTrack(iTrack:=iStation.AccocietedTrack, fPosition:= iStation.PositionOnTrack);
	END_IF
	
	//Add mover to current or found station
	iStation.AddMoverToQueue(iMoverObject);

ELSE
	//Input not valide - ERROR
	SendMoverToGroupExp := E_FAIL;
END_IF
END_METHOD

{attribute 'monitoring':='call'}
PROPERTY StationGroupID : STRING
GET
StationGroupID := THIS^.sStationGroupId;
END_GET
END_PROPERTY

METHOD Update : HRESULT
VAR
	oMover: I_CH_Object;
	iMover: I_XP_MOVER;
	iStation: I_XP_Station;
	pathForFirstMoverInQue: ST_PathFinder;
END_VAR
VAR CONSTANT
	fToleranceMm : LREAL := 1.0; 
END_VAR
//get the first mover in the station queue(the mover at station coordinates)
//all movers are checked here, even those that do not have this station as a destination. Possibly the movers wait in this station until the next station becomes free.
THIS^.fbAssignedMovers.ResetIterator();
WHILE THIS^.fbAssignedMovers.HasNextObject() DO
	IF ToMover(THIS^.fbAssignedMovers.GetNextObject(),iMover) AND_THEN (iMover.HR = S_OK) THEN
			 //Found an mover in this station! Done= Targed reached, PEnding= Moving or an mover in the way
			 // check if first mover has another target than this station. Send away to targed
				IF iMover.TargetStation <> THIS^.StationGroupID AND iMover.TargetStation <> '' THEN
					THIS^.sendMoverToGroupExp(iMover:=iMover, sTargedStationGroupID:= iMover.TargetStation);
				END_IF			 
			 //Exit WHILE Loop
			EXIT;
	END_IF
END_WHILE


Update := S_OK;
END_METHOD

END_FUNCTION_BLOCK

// COMPONENTs/Stationen/I_XP_Station_PLC
INTERFACE I_XP_Station_PLC

{attribute 'monitoring':='call'}
PROPERTY AccocietedTrack : I_XP_Track
GET
END_GET
END_PROPERTY

{attribute 'monitoring':='call'}
PROPERTY Feedback : I_CH_Feedback
GET
END_GET
END_PROPERTY

//Return TRUE if an mover is exactly on the station coordinates and has this station as destination
{attribute 'monitoring':='call'}
PROPERTY IsMoverInStation : BOOL
GET
END_GET
END_PROPERTY

{attribute 'monitoring':='call'}
(* Return interface to mover in station. Return 0 if no mover is in station *)
PROPERTY PlcIfaceToMover : I_XP_Mover_PLC
GET
END_GET
END_PROPERTY

PROPERTY PositionOnTrack : LREAL
GET
END_GET
END_PROPERTY

{attribute 'monitoring':='call'}
PROPERTY PositionXY : REFERENCE TO  PositionXY
GET
END_GET
END_PROPERTY

{attribute 'monitoring':='call'}
PROPERTY Ready : BOOL
GET
END_GET
SET
END_SET
END_PROPERTY

METHOD SendMoverToGroup : I_CH_Feedback
VAR_INPUT 
	sTargedStationGroupID : STRING;
END_VAR
END_METHOD

{attribute 'monitoring':='call'}
PROPERTY StationGroupID : STRING
GET
END_GET
END_PROPERTY

END_INTERFACE

// COMPONENTs/Stationen/FB_XP_Station_FBinit
// The warning " Interface of overridden methode xxx of base I_xxx doesn't match declaration" can be disabled here. 
{warning disable C0094 }
{attribute 'no_explicit_call' := '[FB_ImageSource] Do not call the body - Stick to OOP'}
FUNCTION_BLOCK FB_XP_Station_FBinit EXTENDS FB_XP_Station_Base


{warning restore C0094}

METHOD Configuring : HRESULT
VAR_INPUT
END_VAR
VAR

	fPosOnTrack : LREAL;
	tempPosition : PositionXYC;

END_VAR
Configuring := S_PENDING;
CASE nState_Configuring OF
	0: // Idle
		Configuring := S_OK;
		
	10:	//convert Station position to an valid position on track
		fPosOnTrack := THIS^.iAccocietedTrack.PlanarTrack.GetArcLengthClosestTo(geometry:= THIS^.fbPosition);
		THIS^.iAccocietedTrack.PlanarTrack.GetPositionAt(arcLength:= fPosOnTrack, position:=tempPosition);
		THIS^.fbPosition.SetValuesXY(tempPosition.x, tempPosition.y);
		

		nState_Configuring := 100;


		
   100: // Done
		Configuring := S_OK;
		nState_Configuring := 0;
		
END_CASE

IF fbJsonParser.ExceptionRaised() THEN
	Configuring := E_FAIL;
END_IF

///zzz TODO Errorhandling
END_METHOD

METHOD FB_init : BOOL
VAR_INPUT
	bInitRetains : BOOL; // if TRUE, the retain variables are initialized (warm start / cold start)
	bInCopyCode : BOOL;  // if TRUE, the instance afterwards gets moved into the copy code (online change)
	
	
	oSystem : I_CH_Object;
	
	
	iAccocietedTrack 	: I_XP_Track;//track on which the station is located
	sUniqueIdentification : STRING; //unique identification for this station
	sStationGroupID		: STRING;//to which group of stations does this station belong? e.g. several stations can belong to one 'Infeed' if this is implemented redundantly.
	nCtsMaxMovers 		: UINT;
	xPos, yPos			: LREAL;
	
	//what kind of stations can be reached from this station? several if it has a switch. otherwise it usually only has one
	aStationsAhead1 	: I_CH_Object;
	aStationsAhead2 	: I_CH_Object;
	aStationsAhead3 	: I_CH_Object;
END_VAR

VAR CONSTANT
	MAX_STATION_IN_FRONT : UINT := 3;
END_VAR

VAR 
	nIndex : UINT;
END_VAR
(* Register to the Xplanar System
   1. Test if the interface exists
   2. Test if the object implements a "System for Mover" interface 
*)
IF oSystem <> 0 AND_THEN __QUERYINTERFACE(oSystem,THIS^.iXpSystem) THEN
	THIS^.iXpSystem.RegisterStation(THIS^);
END_IF




THIS^.iAccocietedTrack 	:= iAccocietedTrack;
THIS^.fbSelf.sName		:= sUniqueIdentification;
THIS^.sStationGroupID 	:= sStationGroupID;
THIS^.nCtsMaxMovers 	:= UINT_TO_INT(nCtsMaxMovers);

THIS^.fbPosition.x := xPos;
THIS^.fbPosition.y := yPos;


THIS^.fbStationsAhead.AddObject(iChObject:=aStationsAhead1);
THIS^.fbStationsAhead.AddObject(iChObject:=aStationsAhead2);
THIS^.fbStationsAhead.AddObject(iChObject:=aStationsAhead3);
END_METHOD

END_FUNCTION_BLOCK

// COMPONENTs/Stationen/FB_XP_Station_JSON
// The warning " Interface of overridden methode xxx of base I_xxx doesn't match declaration" can be disabled here. 
{warning disable C0094 }
{attribute 'no_explicit_call' := '[FB_ImageSource] Do not call the body - Stick to OOP'}
FUNCTION_BLOCK FB_XP_Station_JSON  EXTENDS FB_XP_Station_Base
(*
VAR
	{attribute 'hide'}
	bReady 		: BOOL := TRUE;
	{attribute 'hide'}
	sStationGroupID : STRING;
	{attribute 'hide'}
	nCtsMinMovers : INT := 0;
	{attribute 'hide'}
	nCtsMaxMovers : INT := 1;
	{attribute 'hide'}	
	fbPosition : PositionXY;
	{attribute 'hide'}	
	fbJsonParser : FB_JsonDomParser;
	{attribute 'hide'}	
	nState_Configuring: INT;
	{attribute 'hide'}	
	iAccocietedTrack : I_XP_Track;
	{attribute 'hide'}	
	iXpSystem : I_XP_System_Registration;
	
	{attribute 'hide'}
	fbFeedback : FB_CH_Feedback;
	
	(*List of stations*)
	{attribute 'hide'}	
	fbStationsAhead : FB_CH_List;
	
	(* Lists to handle the ownership of movers *)
	{attribute 'hide'}
	fbAssignedMovers 			: FB_CH_List;		// Movers approaching the station

END_VAR
*)
{warning restore C0094}

METHOD Configuring : HRESULT
VAR_INPUT
END_VAR

VAR_INST
    oDocument    : SJsonValue;
	oListOfStations: SJsonValue;
	oListOfStationsAhead: SJsonValue;
	oThisStation : SJsonValue;
	
	
    bExec        : BOOL;

    sPathFull    : STRING;
	
	oItr      : SJsonValue;
    oItrEnd   : SJsonValue;
END_VAR

VAR
    sType      : STRING(10);
	fType 		:LREAL;
	
	iFoundObject : I_CH_Object;
	iTrack : I_XP_Track;

    oProperty : SJsonValue;

	fPosOnTrack : LREAL;
	tempPosition : PositionXYC;

	lrDistMm : LREAL;
END_VAR
Configuring := S_PENDING;
CASE nState_Configuring OF
	0: // Idle
		Configuring := S_OK;
		
	10: // Clear
		// Clear Unique Id
		THIS^.fbSelf.sName := '';
		// delete list of stations ahead
		THIS^.fbStationsAhead.Clear();	
		nState_Configuring := 15;

	15:	// Configure file and load it
		bExec := TRUE;
		sPathFull := XPlanarParameterlist.S_JSON_FOLDER_PATH_ON_TARGED;
		sPathFull := CONCAT(sPathFull,'XP_Stations');
		sPathFull := CONCAT(sPathFull,'.JSON');	
		nState_Configuring := 20;
		
	20: // Load file
		fbJsonParser.LoadDocumentFromFile(sPathFull, bExec);
		IF NOT bExec THEN
			nState_Configuring := 30;
		END_IF
		
	30:	// Loading file		
		oDocument := fbJsonParser.GetDocumentRoot();
		nState_Configuring := 40;
	
	40: // Check file assgnment, load list
		oListOfStations := fbJsonParser.FindMember(oDocument, 'Stations');
	  	IF (oListOfStations <> 0) THEN
		    oItr := fbJsonParser.ArrayBegin(oListOfStations);
		    oItrEnd := fbJsonParser.ArrayEnd(oListOfStations);
			
			nState_Configuring := 50;
		ELSE 
			;//wrong file
	  	END_IF


	50: // Load single segment. Check all station is the Unique ID is already in use, else set it in this station
		IF oItr <> 0 AND_THEN oItrEnd <> 0 AND_THEN oItr <> oItrEnd THEN
			(* Determine segment type *)
			oProperty := fbJsonParser.FindMember(oItr,'LUID');
			sType := fbJsonParser.GetString(oProperty);
			iFoundObject := iXpSystem.Stations.FindLUID(sLUID:=sType);
			IF iFoundObject = 0 THEN
				//not found = this station can use the LUID
				THIS^.fbSelf.sName := sType;
				oThisStation:= oItr;
				nState_Configuring := 70;
			ELSE
				//the LUID is already in use by an other station. try next
				oItr := fbJsonParser.NextArray(oItr);
				nState_Configuring := 50;
			END_IF
		ELSE
		; //End of list. to many stations in PLC
		END_IF	
		
	70: //Writte JSON to Object  -  AccocietedTrack
		oProperty := fbJsonParser.FindMember(oThisStation,'AccocietedTrack');
		sType := fbJsonParser.GetString(oProperty);
		iFoundObject := iXpSystem.Tracks.FindOIDString(sType);
		
		IF iFoundObject <> 0  AND_THEN ToTrack(iFoundObject, iTrack) THEN
			THIS^.iAccocietedTrack := iTrack;
			nState_Configuring := 72;
		ELSE
			;//Error, Track not found			
		END_IF
		
		
	72: //Writte JSON to Object  -  StationGroupId
		oProperty := fbJsonParser.FindMember(oThisStation,'StationGroupId');
		sType := fbJsonParser.GetString(oProperty);
		
		IF sType <> '' THEN
			THIS^.sStationGroupID := sType;
			nState_Configuring := 74;
		ELSE
			;//Error, StationGroupId not found			
		END_IF		
		
	74: //Writte JSON to Object  -  CtsMaxMovers
		oProperty := fbJsonParser.FindMember(oThisStation,'CtsMaxMovers');
		fType := fbJsonParser.GetDouble(oProperty);
		THIS^.nCtsMaxMovers := LREAL_TO_INT(fType);
		nState_Configuring := 76;
		
	76: //Writte JSON to Object  -  Position
		oProperty := fbJsonParser.FindMemberPath(oThisStation,'Position/X');
		fType := fbJsonParser.GetDouble(oProperty);
		tempPosition.x := fType;
		oProperty := fbJsonParser.FindMemberPath(oThisStation,'Position/Y');
		fType := fbJsonParser.GetDouble(oProperty);
		tempPosition.y := fType;
		
		//convert Station position to an valid position on track
		fPosOnTrack := THIS^.iAccocietedTrack.PlanarTrack.GetArcLengthClosestTo(geometry:= tempPosition);
		THIS^.iAccocietedTrack.PlanarTrack.GetPositionAt(arcLength:= fPosOnTrack, position:=tempPosition);
		THIS ^.fbPosition.SetValuesXY(x:=tempPosition.X , y:= tempPosition.Y);

		//check distance between input and calculated point on track. if >50mm, somthing went wrong
		lrDistMm := SQRT(EXPT((tempPosition.x - THIS^.fbPosition.x),2)+EXPT((tempPosition.y - THIS^.fbPosition.y),2));	
		
		IF lrDistMm <= 50.0 THEN
			nState_Configuring := 90;
		ELSE
			;//Error,
		END_IF
		
	90: //wait until all station have an LUID - before linking is not posible
		iFoundObject := iXpSystem.Stations.FindLUID(sLUID:='');
		IF iFoundObject = 0 THEN
			nState_Configuring := 91;
		END_IF
		
	91: // load list of stations ahead
		oListOfStations := fbJsonParser.FindMember(oThisStation, 'StationsAheadIds');
	  	IF (oListOfStations <> 0) THEN
		    oItr := fbJsonParser.ArrayBegin(oListOfStations);
		    oItrEnd := fbJsonParser.ArrayEnd(oListOfStations);
			
			nState_Configuring := 92;
		ELSE 
			;//wrong file
	  	END_IF

	92: // Load single segment. -  StationsAheadIds
		IF oItr <> 0 AND_THEN oItrEnd <> 0 AND_THEN oItr <> oItrEnd THEN
			sType := fbJsonParser.GetString(oItr);
			iFoundObject := iXpSystem.Stations.FindLUID(sLUID:=sType);
			IF iFoundObject <> 0 THEN
				//Add th found station to List
				THIS^.fbStationsAhead.AddObject(iChObject:=iFoundObject);
				//Try next
				oItr := fbJsonParser.NextArray(oItr);
				nState_Configuring := 92;
			ELSE
				; //Error, no station found with this LUID
			END_IF
		ELSE
		//End of list
		nState_Configuring := 100;
		END_IF	
	
		
   100: // Done
		Configuring := S_OK;
		nState_Configuring := 0;
		
END_CASE

IF fbJsonParser.ExceptionRaised() THEN
	Configuring := E_FAIL;
END_IF

///zzz TODO Errorhandling
END_METHOD

METHOD FB_init : BOOL
VAR_INPUT
	bInitRetains : BOOL; // if TRUE, the retain variables are initialized (warm start / cold start)
	bInCopyCode : BOOL;  // if TRUE, the instance afterwards gets moved into the copy code (online change)
	
	
	oSystem : I_CH_Object;
END_VAR
(* Register to the Xplanar System
   1. Test if the interface exists
   2. Test if the object implements a "System for Mover" interface 
*)
IF oSystem <> 0 AND_THEN __QUERYINTERFACE(oSystem,THIS^.iXpSystem) THEN
	THIS^.iXpSystem.RegisterStation(THIS^);
END_IF
END_METHOD

END_FUNCTION_BLOCK

// COMPONENTs/System/FB_XP_System
{attribute 'no_explicit_call' := 'Do not call the body - Stick to OOP'}
FUNCTION_BLOCK FB_XP_System EXTENDS FB_CH_Object IMPLEMENTS I_XP_System_Registration, I_XP_System_PLC
VAR
	{attribute 'hide'}
    fbMovers     : FB_CH_List;
	{attribute 'hide'}	
    fbMoverPairs : FB_CH_List;
	{attribute 'hide'}	
    fbTracks     : FB_CH_List;
	{attribute 'hide'}	
	fbStations 	 : FB_CH_List;
	{attribute 'hide'}	
    iGroup       : I_XP_Group;
	{attribute 'hide'}	
    iEnvironment : I_XP_Environment;
	{attribute 'hide'}
    nState_SEQ_Enabling  : UINT;
	{attribute 'hide'}	
    nState_SEQ_Disabling  : UINT := SEQ_DONE;

	fbFeedback : FB_CH_Feedback;
END_VAR
VAR CONSTANT
	SEQ_DONE : UINT := 999;
END_VAR

METHOD Disable : I_CH_Feedback
VAR_INPUT
END_VAR
//Disable is allways posible

THIS^.nState_SEQ_Disabling 	:= 1;
THIS^.nState_SEQ_Enabling 	:= 0;

THIS^.fbFeedback.LastCommandAccepted:= TRUE;
THIS^.fbFeedback.ActiveCommand 		:= 'Disable';
THIS^.fbFeedback.Busy 				:= TRUE;	
Disable := THIS^.fbFeedback;
END_METHOD

{attribute 'monitoring':='call'}
PROPERTY Disabled : BOOL
GET
Disabled := nState_SEQ_Disabling = SEQ_DONE;
END_GET
END_PROPERTY

METHOD PROTECTED Disabling : HRESULT
VAR
	hr : HRESULT;
	bOk : BOOL := TRUE;
	iTempMover : I_XP_Mover;
	iTempTrack : I_XP_Track;
END_VAR
Disabling := S_PENDING;
CASE nState_SEQ_Disabling OF
	0: // Idle
		Disabling := S_OK;
		
		
	1: // Halt movers
		THIS^.fbMovers.ResetIterator();
		WHILE THIS^.fbMovers.HasNextObject() DO
			IF ToMover(THIS^.fbMovers.GetNextObject(),iTempMover) THEN
				hr := GetMostSignificant(hr, iTempMover.Halt());
			END_IF
		END_WHILE
		
		IF CheckOk(hr) THEN 
			nState_SEQ_Disabling := 20;
		ELSE
			nState_SEQ_Disabling := 1000 + nState_SEQ_Disabling;
		END_IF	
	
		
	20: // Halting movers
		THIS^.fbMovers.ResetIterator();
		WHILE THIS^.fbMovers.HasNextObject() DO
			IF ToMover(THIS^.fbMovers.GetNextObject(),iTempMover) THEN
				bOk := bOk AND iTempMover.PlanarMover.MCTOPLC.SET.SetVelo.x = 0;
				bOk := bOk AND iTempMover.PlanarMover.MCTOPLC.SET.SetVelo.y = 0;
				bOk := bOk AND iTempMover.PlanarMover.MCTOPLC.SET.SetVelo.z = 0;
				bOk := bOk AND iTempMover.PlanarMover.MCTOPLC.SET.SetVelo.a = 0;
				bOk := bOk AND iTempMover.PlanarMover.MCTOPLC.SET.SetVelo.b = 0;
				bOk := bOk AND iTempMover.PlanarMover.MCTOPLC.SET.SetVelo.c = 0;
			END_IF
		END_WHILE
		
		IF bOk THEN 
			nState_SEQ_Disabling := 30;
		END_IF	
		
	
	30: // Reset movers
		THIS^.fbMovers.ResetIterator();
		WHILE THIS^.fbMovers.HasNextObject() DO
			IF ToMover(THIS^.fbMovers.GetNextObject(),iTempMover) THEN
				hr := GetMostSignificant(hr, iTempMover.Reset());
			END_IF
		END_WHILE
		
		IF CheckOk(hr) THEN 
			nState_SEQ_Disabling := 40;
		ELSE
			nState_SEQ_Disabling := 1000 + nState_SEQ_Disabling;
		END_IF		
		
		
	40: // Resetting movers
		THIS^.fbMovers.ResetIterator();
		WHILE THIS^.fbMovers.HasNextObject() DO
			IF ToMover(THIS^.fbMovers.GetNextObject(),iTempMover) THEN
				hr := GetMostSignificant(hr, iTempMover.HR);
			END_IF
		END_WHILE
		
		IF CheckOk(hr) THEN 
			nState_SEQ_Disabling := 50;
		ELSIF FAILED(hr) THEN
			nState_SEQ_Disabling := 1000 + nState_SEQ_Disabling;
		END_IF
		
		
	50: // Disable movers
		THIS^.fbMovers.ResetIterator();
		WHILE THIS^.fbMovers.HasNextObject() DO
			IF ToMover(THIS^.fbMovers.GetNextObject(),iTempMover) THEN
				hr := GetMostSignificant(hr, iTempMover.Disable());
			END_IF
		END_WHILE
		
		IF CheckOk(hr) THEN 
			nState_SEQ_Disabling := 60;
		ELSE
			nState_SEQ_Disabling := 1000 + nState_SEQ_Disabling;
		END_IF			
		
		
	60: // Disabling movers
		THIS^.fbMovers.ResetIterator();
		WHILE THIS^.fbMovers.HasNextObject() DO
			IF ToMover(THIS^.fbMovers.GetNextObject(),iTempMover) THEN
				hr := GetMostSignificant(hr, iTempMover.HR);
			END_IF
		END_WHILE
		
		IF CheckOk(hr) THEN 
			nState_SEQ_Disabling := 61;
		ELSIF FAILED(hr) THEN
			nState_SEQ_Disabling := 1000 + nState_SEQ_Disabling;
		END_IF		


	61: // Reset track
		THIS^.fbTracks.ResetIterator();
		WHILE THIS^.fbTracks.HasNextObject() DO
			IF ToTrack(THIS^.fbTracks.GetNextObject(),iTempTrack) THEN
				hr := GetMostSignificant(hr, iTempTrack.Reset());
			END_IF
		END_WHILE
		
		IF CheckOk(hr) THEN 
			nState_SEQ_Disabling := 62;
		ELSE
			nState_SEQ_Disabling := 1000 + nState_SEQ_Disabling;
		END_IF		
		
		
	62: // Resetting track
		THIS^.fbTracks.ResetIterator();
		WHILE THIS^.fbTracks.HasNextObject() DO
			IF ToTrack(THIS^.fbTracks.GetNextObject(),iTempTrack) THEN
				hr := GetMostSignificant(hr, iTempTrack.HR);
			END_IF
		END_WHILE
		
		IF CheckOk(hr) THEN 
			nState_SEQ_Disabling := 63;
		ELSIF FAILED(hr) THEN
			nState_SEQ_Disabling := 1000 + nState_SEQ_Disabling;
		END_IF	

				
	63: // Reset group
		hr := iGroup.Reset();
		
		IF CheckOk(hr) THEN 
			nState_SEQ_Disabling := 64;
		ELSE
			nState_SEQ_Disabling := 1000 + nState_SEQ_Disabling;
		END_IF		
		
		
	64: // Resetting group
		hr := iGroup.HR;
		
		IF CheckOk(hr) THEN 
			nState_SEQ_Disabling := 70;
		ELSIF FAILED(hr) THEN
			nState_SEQ_Disabling := 1000 + nState_SEQ_Disabling;
		END_IF		
		
		
		

   70: // Disable tracks
		THIS^.fbTracks.ResetIterator();
		WHILE THIS^.fbTracks.HasNextObject() DO
			IF ToTrack(THIS^.fbTracks.GetNextObject(),iTempTrack) THEN
				hr := GetMostSignificant(hr, iTempTrack.Disable());
			END_IF
		END_WHILE
		
		IF CheckOk(hr) THEN 
			nState_SEQ_Disabling := 80;
		ELSE
			nState_SEQ_Disabling := 1000 + nState_SEQ_Disabling;
		END_IF			
   
		
   80: // Disabling tracks
		THIS^.fbTracks.ResetIterator();
		WHILE THIS^.fbTracks.HasNextObject() DO
			IF ToTrack(THIS^.fbTracks.GetNextObject(),iTempTrack) THEN
				hr := GetMostSignificant(hr, iTempTrack.HR);
			END_IF
		END_WHILE
		
		IF CheckOk(hr) THEN 
			nState_SEQ_Disabling := 90;
		ELSIF FAILED(hr) THEN
			nState_SEQ_Disabling := 1000 + nState_SEQ_Disabling;
		END_IF	
				

	90: // Disable group
		hr := iGroup.Disable();
		
		IF CheckOk(hr) THEN 
			nState_SEQ_Disabling := 100;
		ELSE
			nState_SEQ_Disabling := 1000 + nState_SEQ_Disabling;
		END_IF	
		
		
   100: // Disabling group
		hr := iGroup.HR;
		
		IF CheckOk(hr) THEN 
			nState_SEQ_Disabling := 105;
		ELSIF FAILED(hr) THEN
			nState_SEQ_Disabling := 1000 + nState_SEQ_Disabling;
		END_IF	

		
  105: // Remove tracks from group
		THIS^.fbTracks.ResetIterator();
		WHILE THIS^.fbTracks.HasNextObject() DO
			IF ToTrack(THIS^.fbTracks.GetNextObject(),iTempTrack) THEN
				hr := GetMostSignificant(hr, iTempTrack.RemoveFromGroup());
			END_IF
		END_WHILE
		
		IF CheckOk(hr) THEN 
			nState_SEQ_Disabling := 106;
		ELSE
			nState_SEQ_Disabling := 1000 + nState_SEQ_Disabling;
		END_IF			
   
		
   106: // Removing tracks from group
		THIS^.fbTracks.ResetIterator();
		WHILE THIS^.fbTracks.HasNextObject() DO
			IF ToTrack(THIS^.fbTracks.GetNextObject(),iTempTrack) THEN
				bOk := bOk AND iTempTrack.PlanarTrack.MCTOPLC_STD.GroupOID = 0;
			END_IF
		END_WHILE
		
		IF bOk THEN 
			nState_SEQ_Disabling := 110;
		END_IF	
		
		
	110: // Remove movers from group
		THIS^.fbMovers.ResetIterator();
		WHILE THIS^.fbMovers.HasNextObject() DO
			IF ToMover(THIS^.fbMovers.GetNextObject(),iTempMover) THEN
				hr := GetMostSignificant(hr, iTempMover.RemoveFromGroup());
			END_IF
		END_WHILE
		
		IF CheckOk(hr) THEN 
			nState_SEQ_Disabling := 120;
		ELSE
			nState_SEQ_Disabling := 1000 + nState_SEQ_Disabling;
		END_IF		
	
		
	120: // Removing movers from group
		THIS^.fbMovers.ResetIterator();
		WHILE THIS^.fbMovers.HasNextObject() DO
			IF ToMover(THIS^.fbMovers.GetNextObject(),iTempMover) THEN
				bOk := bOk AND iTempMover.PlanarMover.MCTOPLC.STD.GroupOID = 0;
			END_IF
		END_WHILE
		
		IF bOk THEN 
			nState_SEQ_Disabling := 130;
		END_IF		
	
		
	130: // Remove envirement from group
		hr := iEnvironment.RemoveFromGroup();
		
		IF CheckOk(hr) THEN 
			nState_SEQ_Disabling := 140;
		ELSE
			nState_SEQ_Disabling := 1000 + nState_SEQ_Disabling;
		END_IF		
		
		
   140: // Removing envirement from group
		//IF CheckOk(iEnvironment.HR) OR (iEnvironment.Self.MCTOPLC_STD.GroupOID = 0) THEN 
		hr := iEnvironment.HR;
	
		IF CheckOk(hr) THEN 
			nState_SEQ_Disabling := SEQ_DONE;
		ELSIF FAILED(hr) THEN
			nState_SEQ_Disabling := 1000 + nState_SEQ_Disabling;
		END_IF	
		
(*23.08.2023 do not .Clear(). This will delete the stators config.
 		
   150: // Clear environment
		hr := iEnvironment.Clear();
		
		IF CheckOk(hr) THEN 
			nState_SEQ_Disabling := 160;
		ELSE
			nState_SEQ_Disabling := 1000 + nState_SEQ_Disabling;
		END_IF	
		
	
   160: // Clearing environment (delete boundary)
		hr := (iEnvironment.HR);
		IF CheckOk(hr) THEN 
			nState_SEQ_Disabling := SEQ_DONE;
		ELSIF FAILED(hr) THEN
			nState_SEQ_Disabling := 1000 + nState_SEQ_Disabling;
		END_IF	 
*)		
	
   SEQ_DONE: //Done
   		Disabling := S_OK;

		
	1000..1999://Error
		hr := GetMostSignificant(hr, E_FAIL);

END_CASE

// Propagate error
IF FAILED(hr) THEN
	Disabling := hr;
END_IF
END_METHOD

METHOD Enable : I_CH_Feedback
VAR_INPUT
END_VAR
IF NOT THIS^.fbFeedback.Done THEN
	//Error active/not ready
	THIS^.fbFeedback.LastCommandAccepted 	:= FALSE;

ELSIF nState_SEQ_Enabling <> 0 THEN
	//System is partial or full enabled. Disable first.
	THIS^.fbFeedback.LastCommandAccepted 	:= FALSE;
ELSE
	THIS^.nState_SEQ_Disabling 	:= 0;
	THIS^.nState_SEQ_Enabling 	:= 1;
	THIS^.fbFeedback.LastCommandAccepted 	:= TRUE;
	THIS^.fbFeedback.ActiveCommand 			:= 'Enable';
	THIS^.fbFeedback.Busy 				 	:= TRUE;	
END_IF

Enable := THIS^.fbFeedback;
END_METHOD

{attribute 'monitoring':='call'}
PROPERTY Enabled : BOOL
GET
Enabled := nState_SEQ_Enabling = SEQ_DONE;
END_GET
END_PROPERTY

METHOD PROTECTED Enabling : HRESULT
VAR
	hr : HRESULT;
	
	iTempMover : I_XP_Mover;
	iTempMoverPair : I_XP_MoverPair;
	iTempStation : I_XP_Station;
	iTempTrack : I_XP_Track;
	
	lrCRotationShortestPos : LREAL;
END_VAR

VAR_INST
	fbTimeOutSeq : TON; 
END_VAR
Enabling := S_PENDING;
CASE nState_SEQ_Enabling OF
	0: // Idle
		Enabling := S_OK;	
		
	1: //Redetect all movers on real system
		IF THIS^.iEnvironment.UtilityEnvirement.XpuTcIo(1).GetOperationMode() = OperationMode.Normal THEN
			THIS^.iEnvironment.UtilityEnvirement.XpuTcIo(1).SetStartMoverRedetection();	
		END_IF
		nState_SEQ_Enabling := 5;

		
	5: //Compare detectet and expectet movers	
	   //timeout is monitored in this sequence
		IF (THIS^.iEnvironment.UtilityEnvirement.XpuTcIo(1).GetMoverDetectionInfos().APM4220Detected = THIS^.iEnvironment.UtilityEnvirement.XpuTcIo(1).GetMoverDetectionInfos().APM4220Expected AND
			THIS^.iEnvironment.UtilityEnvirement.XpuTcIo(1).GetMoverDetectionInfos().APM4221Detected = THIS^.iEnvironment.UtilityEnvirement.XpuTcIo(1).GetMoverDetectionInfos().APM4221Expected AND
			THIS^.iEnvironment.UtilityEnvirement.XpuTcIo(1).GetMoverDetectionInfos().APM4330Detected = THIS^.iEnvironment.UtilityEnvirement.XpuTcIo(1).GetMoverDetectionInfos().APM4330Expected AND
			THIS^.iEnvironment.UtilityEnvirement.XpuTcIo(1).GetMoverDetectionInfos().APM4550Detected = THIS^.iEnvironment.UtilityEnvirement.XpuTcIo(1).GetMoverDetectionInfos().APM4550Expected AND
			THIS^.iEnvironment.UtilityEnvirement.XpuTcIo(1).GetMoverDetectionInfos().TotalDetected   = THIS^.iEnvironment.UtilityEnvirement.XpuTcIo(1).GetMoverDetectionInfos().TotalExpected 	
		   )THEN
			nState_SEQ_Enabling := 10;
		END_IF	
			
		
	10: // Reset movers
		THIS^.fbMovers.ResetIterator();
		WHILE THIS^.fbMovers.HasNextObject() DO
			IF ToMover(THIS^.fbMovers.GetNextObject(),iTempMover) THEN
				hr := GetMostSignificant(hr, iTempMover.Reset());
			END_IF
		END_WHILE
		
		IF CheckOk(hr) THEN 
			nState_SEQ_Enabling := 20;
		ELSE
			nState_SEQ_Enabling := 1000 + nState_SEQ_Enabling;
		END_IF		
		
		
	20: // Resetting movers
		THIS^.fbMovers.ResetIterator();
		WHILE THIS^.fbMovers.HasNextObject() DO
			IF ToMover(THIS^.fbMovers.GetNextObject(),iTempMover) THEN
				hr := GetMostSignificant(hr, iTempMover.HR);
			END_IF
		END_WHILE
		
		IF CheckOk(hr) THEN 
			nState_SEQ_Enabling := 25;
		ELSIF FAILED(hr) THEN
			nState_SEQ_Enabling := 1000 + nState_SEQ_Enabling;
		END_IF

	25:// Build pairs
		(* Reset the iterators*)
		THIS^.fbMovers.ResetIterator();
		THIS^.fbMoverPairs.ResetIterator();
		
		(* For each pair *)
		WHILE THIS^.fbMoverPairs.HasNextObject() DO
			(* IF the pair is valid *)
			IF ToMoverPair(THIS^.fbMoverPairs.GetNextObject(), iTempMoverPair) THEN
				(* Assign a master mover to it *)
				IF THIS^.fbMovers.HasNextObject() AND_THEN ToMover(THIS^.fbMovers.GetNextObject(),iTempMover) THEN
					iTempMoverPair.MoverMaster := iTempMover;
				END_IF
				(* Assign a slave mover to it *)
				IF THIS^.fbMovers.HasNextObject() AND_THEN ToMover(THIS^.fbMovers.GetNextObject(),iTempMover) THEN
					iTempMoverPair.MoverSlave := iTempMover;
				END_IF
			END_IF
		END_WHILE
		nState_SEQ_Enabling := 30;	
		
	30: // Configure environment
		hr := iEnvironment.Configure();
		
		IF CheckOk(hr) THEN 
			nState_SEQ_Enabling := 40;
		ELSE
			nState_SEQ_Enabling := 1000 + nState_SEQ_Enabling;
		END_IF	
	
	40: // Configuring environment
		hr := iEnvironment.HR;
		
		IF CheckOk(hr) THEN 
			nState_SEQ_Enabling := 50;
		ELSIF FAILED(hr) THEN
			nState_SEQ_Enabling := 1000 + nState_SEQ_Enabling;
		END_IF
		
	50: // Add environment to group
		hr := iEnvironment.AddToGroup(iGroup);
		
		IF CheckOk(hr) THEN 
			nState_SEQ_Enabling := 60;
		ELSE
			nState_SEQ_Enabling := 1000 + nState_SEQ_Enabling;
		END_IF		
	
	60: // Adding environment to group
		hr := iEnvironment.HR;
		
		IF CheckOk(hr) THEN 
			nState_SEQ_Enabling := 70;
		ELSIF FAILED(hr) THEN
			nState_SEQ_Enabling := 1000 + nState_SEQ_Enabling;
		END_IF

	70: // Configure the tracks |
		THIS^.fbTracks.ResetIterator();
		WHILE THIS^.fbTracks.HasNextObject() DO
			IF ToTrack(THIS^.fbTracks.GetNextObject(),iTempTrack) THEN
				hr := GetMostSignificant(hr, iTempTrack.Configure());
			END_IF
		END_WHILE
		
		IF CheckOk(hr) THEN 
			nState_SEQ_Enabling := 71;
		ELSE
			nState_SEQ_Enabling := 1000 + nState_SEQ_Enabling;
		END_IF	
		
		
	71: // Configuring the tracks 
		THIS^.fbTracks.ResetIterator();
		WHILE THIS^.fbTracks.HasNextObject() DO
			IF ToTrack(THIS^.fbTracks.GetNextObject(),iTempTrack) THEN
				hr := GetMostSignificant(hr, iTempTrack.Configuring());
			END_IF
		END_WHILE
		
		IF CheckOk(hr) THEN 
			nState_SEQ_Enabling := 80;
		ELSIF FAILED(hr) THEN
			nState_SEQ_Enabling := 1000 + nState_SEQ_Enabling;
		END_IF	
		
	80: // Enable the tracks
		THIS^.fbTracks.ResetIterator();
		WHILE THIS^.fbTracks.HasNextObject() DO
			IF ToTrack(THIS^.fbTracks.GetNextObject(),iTempTrack) THEN
				hr := GetMostSignificant(hr, iTempTrack.Enable());
			END_IF
		END_WHILE
		
		IF CheckOk(hr) THEN 
			nState_SEQ_Enabling := 90;
		ELSE
			nState_SEQ_Enabling := 1000 + nState_SEQ_Enabling;
		END_IF		
	
	90: // Enabling the tracks
		THIS^.fbTracks.ResetIterator();
		WHILE THIS^.fbTracks.HasNextObject() DO
			IF ToTrack(THIS^.fbTracks.GetNextObject(),iTempTrack) THEN
				hr := GetMostSignificant(hr, iTempTrack.HR);
			END_IF
		END_WHILE
		
		IF CheckOk(hr) THEN 
			nState_SEQ_Enabling := 95;
		ELSIF FAILED(hr) THEN
			nState_SEQ_Enabling := 1000 + nState_SEQ_Enabling;
		END_IF	
		
	95: // Add tracks to group
		THIS^.fbTracks.ResetIterator();
		WHILE THIS^.fbTracks.HasNextObject() DO
			IF ToTrack(THIS^.fbTracks.GetNextObject(),iTempTrack) THEN
				hr := GetMostSignificant(hr, iTempTrack.AddToGroup(iGroup));
			END_IF
		END_WHILE
		
		IF CheckOk(hr) THEN 
			nState_SEQ_Enabling := 96;
		ELSE
			nState_SEQ_Enabling := 1000 + nState_SEQ_Enabling;
		END_IF	

	96: // Adding tracks to group
		THIS^.fbTracks.ResetIterator();
		WHILE THIS^.fbTracks.HasNextObject() DO
			IF ToTrack(THIS^.fbTracks.GetNextObject(),iTempTrack) THEN
				hr := GetMostSignificant(hr, iTempTrack.HR);
			END_IF
		END_WHILE
		
		IF CheckOk(hr) THEN 
			nState_SEQ_Enabling := 100;
		ELSIF FAILED(hr) THEN
			nState_SEQ_Enabling := 1000 + nState_SEQ_Enabling;
		END_IF		
			
   100: // Calculate track trace
		THIS^.fbTracks.ResetIterator();
		WHILE THIS^.fbTracks.HasNextObject() DO
			IF ToTrack(THIS^.fbTracks.GetNextObject(),iTempTrack) THEN
				hr := GetMostSignificant(hr, iTempTrack.CalcTrackPoints());
			END_IF
		END_WHILE
		
		IF CheckOk(hr) THEN 
			nState_SEQ_Enabling := 102;
		ELSE
			nState_SEQ_Enabling := 1000 + nState_SEQ_Enabling;
		END_IF
	
	102: // Config Station
		THIS^.fbStations.ResetIterator();
		WHILE THIS^.fbStations.HasNextObject() DO
			IF ToStation(THIS^.fbStations.GetNextObject(),iTempStation) THEN
				hr := GetMostSignificant(hr, iTempStation.Configure());
			END_IF
		END_WHILE
		
		IF CheckOk(hr) THEN 
			nState_SEQ_Enabling := 103;
		ELSE
			nState_SEQ_Enabling := 1000 + nState_SEQ_Enabling;
		END_IF		
		
	103: // Configuring Stations
		THIS^.fbStations.ResetIterator();
		WHILE THIS^.fbStations.HasNextObject() DO
			IF ToStation(THIS^.fbStations.GetNextObject(),iTempStation) THEN
				hr := GetMostSignificant(hr, iTempStation.Configuring());
			END_IF
		END_WHILE
		
		IF CheckOk(hr) THEN 
			nState_SEQ_Enabling := 110;
		ELSIF FAILED(hr) THEN
			nState_SEQ_Enabling := 1000 + nState_SEQ_Enabling;
		END_IF	
		
		
	110: // Enable movers
		THIS^.fbMovers.ResetIterator();
		WHILE THIS^.fbMovers.HasNextObject() DO
			IF ToMover(THIS^.fbMovers.GetNextObject(),iTempMover) THEN
				hr := GetMostSignificant(hr, iTempMover.Enable());
			END_IF
		END_WHILE
		
		IF CheckOk(hr) THEN 
			nState_SEQ_Enabling := 120;
		ELSE
			nState_SEQ_Enabling := 1000 + nState_SEQ_Enabling;
		END_IF	
		
	120: // Enabling movers
		THIS^.fbMovers.ResetIterator();
		WHILE THIS^.fbMovers.HasNextObject() DO
			IF ToMover(THIS^.fbMovers.GetNextObject(),iTempMover) THEN
				hr := GetMostSignificant(hr, iTempMover.HR);
			END_IF
		END_WHILE
		
		IF CheckOk(hr) THEN 
			nState_SEQ_Enabling := 122;
		ELSIF FAILED(hr) THEN
			nState_SEQ_Enabling := 1000 + nState_SEQ_Enabling;
		END_IF	

	122: //Rotate C-Axis to "Zero" (to the next 90 degree pitch)
		THIS^.fbMovers.ResetIterator();
		WHILE THIS^.fbMovers.HasNextObject() DO
			IF ToMover(THIS^.fbMovers.GetNextObject(),iTempMover) THEN
				// Decide which 90 degree pitch is closer to the current position. If the remainder is greater than 45 degrees, then round up to the next 90 degree division.
				lrCRotationShortestPos := LREAL_TO_DINT(lrCRotationShortestPos / 90.0) * 90.0;
				hr := GetMostSignificant(hr, iTempMover.MoveC(lrCRotationShortestPos));
			END_IF
		END_WHILE
		
		IF CheckOk(hr) THEN 
			nState_SEQ_Enabling := 123;
		ELSE
			nState_SEQ_Enabling := 1000 + nState_SEQ_Enabling;
		END_IF	
		
	123: //Rotating C-Axis to Zero			
		THIS^.fbMovers.ResetIterator();
		WHILE THIS^.fbMovers.HasNextObject() DO
			IF ToMover(THIS^.fbMovers.GetNextObject(),iTempMover) THEN
				hr := GetMostSignificant(hr, iTempMover.HR);
			END_IF
		END_WHILE
		
		IF CheckOk(hr) THEN 
			nState_SEQ_Enabling := 130;
		ELSIF FAILED(hr) THEN
			nState_SEQ_Enabling := 1000 + nState_SEQ_Enabling;
		END_IF	
		
	130: // Add movers to group
		THIS^.fbMovers.ResetIterator();
		WHILE THIS^.fbMovers.HasNextObject() DO
			IF ToMover(THIS^.fbMovers.GetNextObject(),iTempMover) THEN
				hr := GetMostSignificant(hr, iTempMover.AddToGroup(THIS^.iGroup));
			END_IF
		END_WHILE
		
		IF CheckOk(hr) THEN 
			nState_SEQ_Enabling := 140;
		ELSE
			nState_SEQ_Enabling := 1000 + nState_SEQ_Enabling;
		END_IF	
	
	140: // Adding mover to group
		THIS^.fbMovers.ResetIterator();
		WHILE THIS^.fbMovers.HasNextObject() DO
			IF ToMover(THIS^.fbMovers.GetNextObject(),iTempMover) THEN
				hr := GetMostSignificant(hr, iTempMover.HR);
			END_IF
		END_WHILE
		
		IF CheckOk(hr) THEN 
			nState_SEQ_Enabling := 150;
		ELSIF FAILED(hr) THEN
			nState_SEQ_Enabling := 1000 + nState_SEQ_Enabling;
		END_IF		
	
	150: // Enable group
		hr := iGroup.Enable();
		
		IF CheckOk(hr) THEN 
			nState_SEQ_Enabling := 160;
		ELSE
			nState_SEQ_Enabling := 1000 + nState_SEQ_Enabling;
		END_IF	
		
	160: // Enabling group
		hr := iGroup.HR;
		
		IF CheckOk(hr) THEN 
			nState_SEQ_Enabling := 170;
		ELSIF FAILED(hr) THEN
			nState_SEQ_Enabling := 1000 + nState_SEQ_Enabling;
		END_IF	

	170: // Waiting movers are in free movement
		THIS^.fbMovers.ResetIterator();
		WHILE THIS^.fbMovers.HasNextObject() DO
			IF ToMover(THIS^.fbMovers.GetNextObject(),iTempMover) THEN
				hr := GetMostSignificant(hr, iTempMover.HR);
				IF NOT (iTempMover.Mode = MC_PLANAR_MOVER_COMMAND_MODE.FreeMovement) THEN
					hr := GetMostSignificant(hr, S_PENDING);
				END_IF
			END_IF
		END_WHILE
		
		IF CheckOk(hr) THEN 
			nState_SEQ_Enabling := 180;
		ELSIF FAILED(hr) THEN
			nState_SEQ_Enabling := 1000 + nState_SEQ_Enabling;
		END_IF	
				
	180: // Join the track on startup. outsourced to a method for easier overwriting
		IF NOT fbTracks.IsEmpty THEN
			hr := THIS^.JoiningTrack(); 
		END_IF

		
		IF CheckOk(hr) THEN 
			nState_SEQ_Enabling := 190;
		ELSIF FAILED(hr) THEN
			nState_SEQ_Enabling := 1000 + nState_SEQ_Enabling;
		END_IF	

		
	190: // Joining closest track check feedback
		IF NOT fbTracks.IsEmpty THEN
			THIS^.fbMovers.ResetIterator();
			WHILE THIS^.fbMovers.HasNextObject() DO
				IF ToMover(THIS^.fbMovers.GetNextObject(),iTempMover) THEN
					hr := GetMostSignificant(hr, iTempMover.HR);
					IF NOT (iTempMover.Mode = MC_PLANAR_MOVER_COMMAND_MODE.OnTrack) THEN
						hr := GetMostSignificant(hr, S_PENDING);
					END_IF
				END_IF
			END_WHILE
		END_IF
		
		IF CheckOk(hr) THEN 
			nState_SEQ_Enabling := 200;
		ELSIF FAILED(hr) THEN
			nState_SEQ_Enabling := 1000 + nState_SEQ_Enabling;
		END_IF	

		
	200: // Distribute the movers to the available stations.
		 // outsourced to a method for easier overwriting
		 IF NOT fbStations.IsEmpty THEN
			 hr := THIS^.JoiningStation();
		 END_IF
		

		IF CheckOk(hr) THEN 
			nState_SEQ_Enabling := SEQ_DONE;
		ELSIF FAILED(hr) THEN
			nState_SEQ_Enabling := 1000 + nState_SEQ_Enabling;
		END_IF	

		
	SEQ_DONE: // Done
		Enabling := S_OK;

		
	1000..1999://Error
		hr := GetMostSignificant(hr, E_FAIL);
END_CASE


//Timeout after to long stay in one of the following seq.
fbTimeOutSeq.IN := (nState_SEQ_Enabling = 5);
fbTimeOutSeq.PT := T#5S;
fbTimeOutSeq();

IF fbTimeOutSeq.Q THEN
	//next seq is error
	nState_SEQ_Enabling := 1000 + nState_SEQ_Enabling;
END_IF


// Propagate error
IF FAILED(hr) THEN
	Enabling := hr;
END_IF
END_METHOD

METHOD Station : I_XP_Station_PLC
VAR_INPUT
	sLUID : STRING;
END_VAR
//IF no station was found, INTERFACE is 0 -> can generate fatal error
__QUERYINTERFACE(THIS^.fbStations.FindLUID(sLUID),Station);
END_METHOD

//Return TRUE if unique station id is valid. if false, interfacepointer is zero -> fatal error
METHOD ValidLUID : BOOL
VAR_INPUT
	sLUID : STRING;
END_VAR
VAR
	iTempInterface : I_XP_Station_PLC;
END_VAR
iTempInterface := THIS^.Station(sLUID := sLUID);
ValidLUID := (iTempInterface <> 0);
END_METHOD

METHOD LinkEnvironment : HRESULT
VAR_INPUT
	oEnvironment : I_CH_Object;
END_VAR

VAR
	iXpEnvironment : I_XP_Environment;
END_VAR
IF oEnvironment <> 0 AND_THEN __QUERYINTERFACE(oEnvironment,iXpEnvironment) THEN
	THIS^.iEnvironment := iXpEnvironment;
END_IF
END_METHOD

METHOD LinkGroup : HRESULT
VAR_INPUT
	oGroup : I_CH_Object;
END_VAR

VAR
	iXpGroup : I_XP_Group;
END_VAR
IF oGroup <> 0 AND_THEN __QUERYINTERFACE(oGroup,iXpGroup) THEN
	THIS^.iGroup := iXpGroup;
END_IF
END_METHOD

METHOD RegisterMover : HRESULT
VAR_INPUT
	oMover : I_CH_Object;
END_VAR

VAR
	iXpMover : I_XP_Mover;
END_VAR
IF oMover <> 0 AND_THEN __QUERYINTERFACE(oMover,iXpMover) THEN
	THIS^.fbMovers.AddObject(oMover);
END_IF
END_METHOD

METHOD RegisterMoverPair : HRESULT
VAR_INPUT
	oMoverPair : I_CH_Object;
END_VAR

VAR
	iXpMoverPair : I_XP_MoverPair;
END_VAR
IF oMoverPair <> 0 AND_THEN __QUERYINTERFACE(oMoverPair,iXpMoverPair) THEN
	THIS^.fbMoverPairs.AddObject(oMoverPair);
END_IF
END_METHOD

METHOD RegisterStation : HRESULT
VAR_INPUT
	oStation : I_CH_Object;
END_VAR

VAR
	iStation : I_XP_Station;
END_VAR
IF oStation <> 0 AND_THEN __QUERYINTERFACE(oStation,iStation) THEN
	THIS^.fbStations.AddObject(oStation);
END_IF
END_METHOD

METHOD RegisterTrack : HRESULT
VAR_INPUT
	oTrack : I_CH_Object;
END_VAR

VAR
	iXpTrack : I_XP_Track;
END_VAR
IF oTrack <> 0 AND_THEN __QUERYINTERFACE(oTrack,iXpTrack) THEN
	THIS^.fbTracks.AddObject(oTrack);
END_IF
END_METHOD

METHOD PROTECTED JoiningStation : HRESULT
VAR_INPUT
END_VAR
VAR
	hr : HRESULT;
	iTempMover : I_XP_Mover;
	iTempStation : I_XP_Station;
END_VAR
//remove all movers from stations
THIS^.fbStations.ResetIterator();	
WHILE THIS^.fbStations.HasNextObject() DO
	IF ToStation(THIS^.fbStations.GetNextObject(),iTempStation) THEN
		hr := GetMostSignificant(hr, iTempStation.DeleteMoversQueue());
	END_IF	
END_WHILE

//Move all movers to station 1. This is only working if station 1 can store so many movers.
THIS^.fbMovers.ResetIterator();
THIS^.fbStations.ResetIterator();		
IF ToStation(THIS^.fbStations.GetNextObject(),iTempStation) THEN
	WHILE THIS^.fbMovers.HasNextObject() DO
		ToMover(THIS^.fbMovers.GetNextObject(),iTempMover);
		hr := GetMostSignificant(hr, iTempStation.sendMoverToGroupExp(sTargedStationGroupID:=iTempStation.StationGroupID, iMover:= iTempMover));
	END_WHILE
END_IF


//In this strategy all movers need to move to station 1. If hr is not 0, then station was not found or is full
IF CheckNotOk(hr) THEN 
	JoiningStation := GetMostSignificant(hr, E_FAIL);
ELSE
	JoiningStation := S_OK;
END_IF
END_METHOD

METHOD PROTECTED JoiningTrack : HRESULT
VAR	
	hr : HRESULT;
	iClosestTrack : I_XP_Track;	
	iTempMover : I_XP_Mover;
	iTempTrack : I_XP_Track;
	fDistance : LREAL;
	fShortestDistance : LREAL;
END_VAR

VAR CONSTANT
	MAX_LREAL_VALUE: LREAL := 1.7976931348623158E+308;
END_VAR
JoiningTrack := S_PENDING;

// Join closest track
THIS^.fbMovers.ResetIterator();
WHILE THIS^.fbMovers.HasNextObject() DO
	IF ToMover(THIS^.fbMovers.GetNextObject(),iTempMover) THEN
		
		//check all track to decide which is the closest
		THIS^.fbTracks.ResetIterator();
		fShortestDistance := MAX_LREAL_VALUE;
		WHILE THIS^.fbTracks.HasNextObject() DO
			IF ToTrack(THIS^.fbTracks.GetNextObject(),iTempTrack) THEN
				fDistance := iTempMover.DistToTrack(iTempTrack);
				//closer track found
				IF fDistance <= fShortestDistance THEN
					iClosestTrack := iTempTrack;
					fShortestDistance := fDistance;
				END_IF
			END_IF
		END_WHILE
		
		//send mover to found closest track
		IF iClosestTrack <> 0 THEN
			hr := GetMostSignificant(hr, iTempMover.JoinTrack(iClosestTrack));
		ELSE
			hr := GetMostSignificant(hr, E_FAIL);
		END_IF
	END_IF
END_WHILE

IF FAILED(hr) THEN 
	JoiningTrack := hr;
ELSE	
	JoiningTrack := S_OK;
END_IF

JoiningTrack := hr;
END_METHOD

PROPERTY Enviroment : I_XP_Environment
GET
Enviroment := THIS^.iEnvironment;
END_GET
END_PROPERTY

{attribute 'monitoring':='call'}
PROPERTY Feedback : I_CH_Feedback
GET
Feedback := THIS^.fbFeedback;
END_GET
END_PROPERTY

METHOD Initialize : HRESULT
VAR_INPUT
END_VAR
VAR
	hr : HRESULT;
END_VAR
hr := S_OK;


hr := GetMostSignificant(hr, THIS^.fbMovers.Initialize());
hr := GetMostSignificant(hr, THIS^.fbMoverPairs.Initialize());
hr := GetMostSignificant(hr, THIS^.fbTracks.Initialize());
hr := GetMostSignificant(hr, THIS^.fbStations.Initialize());
hr := GetMostSignificant(hr, THIS^.iEnvironment.Initialize());
hr := GetMostSignificant(hr, THIS^.iGroup.Initialize());



Initialize := hr;
END_METHOD

PROPERTY Movers : I_CH_LIST
GET
Movers := THIS^.fbMovers;
END_GET
END_PROPERTY

PROPERTY Stations : I_CH_LIST
GET
Stations := THIS^.fbStations;
END_GET
END_PROPERTY

PROPERTY Tracks : I_CH_LIST
GET
Tracks := THIS^.fbTracks;
END_GET
END_PROPERTY

METHOD Update : HRESULT
VAR_INPUT
END_VAR
VAR
	hr : HRESULT;
END_VAR
hr := S_OK;


hr := GetMostSignificant(hr, THIS^.Enabling());
hr := GetMostSignificant(hr, THIS^.Disabling());

THIS^.fbFeedback.HR := hr;


hr := GetMostSignificant(hr, THIS^.fbMovers.Update());
hr := GetMostSignificant(hr, THIS^.fbMoverPairs.Update());
hr := GetMostSignificant(hr, THIS^.fbTracks.Update());
hr := GetMostSignificant(hr, THIS^.fbStations.Update());
hr := GetMostSignificant(hr, THIS^.iGroup.Update());
hr := GetMostSignificant(hr, THIS^.iEnvironment.Update());


Update:= hr;
END_METHOD

END_FUNCTION_BLOCK

// COMPONENTs/System/I_XP_System_PLC
INTERFACE I_XP_System_PLC EXTENDS I_CH_Object

METHOD Disable : I_CH_Feedback
VAR_INPUT
END_VAR
END_METHOD

{attribute 'monitoring':='call'}
PROPERTY Disabled : BOOL
GET
END_GET
END_PROPERTY

METHOD Enable : I_CH_Feedback
VAR_INPUT
END_VAR
END_METHOD

{attribute 'monitoring':='call'}
PROPERTY Enabled : BOOL
GET
END_GET
END_PROPERTY

{attribute 'monitoring':='call'}
PROPERTY Feedback : I_CH_Feedback
GET
END_GET
END_PROPERTY

METHOD Initialize : HRESULT
VAR_INPUT
END_VAR
END_METHOD

METHOD Station : I_XP_Station_PLC
VAR_INPUT
	sLUID : STRING;
END_VAR
END_METHOD

METHOD Update : HRESULT
VAR_INPUT
END_VAR
END_METHOD

//Return TRUE if unique station id is valid. if false, interfacepointer is zero -> fatal error
METHOD ValidLUID : BOOL
VAR_INPUT
	sLUID : STRING;
END_VAR
END_METHOD

END_INTERFACE

// COMPONENTs/Track/FB_XP_Track_Base
{attribute 'no_explicit_call' := '[FB_ImageSource] Do not call the body - Stick to OOP'}
FUNCTION_BLOCK ABSTRACT FB_XP_Track_Base EXTENDS FB_CH_Object IMPLEMENTS I_XP_Track
VAR
	fbActiveCmd : MC_PlanarFeedback;	

	fbTrack : MC_PlanarTrack;
	{attribute 'hide'}
	iXpSystem : I_XP_System_Registration;
	{attribute 'hide'}	
	nState_Configuring : UINT;
	
	afTrackPoints		: ARRAY[0..XplanarParameterlist.N_TRACE_POINTS] OF PositionXYC;
END_VAR

METHOD AddToGroup : HRESULT
VAR_INPUT
	iGroup : I_XP_Group;
END_VAR
IF NOT THIS^.fbActiveCmd.Busy AND NOT THIS^.fbActiveCmd.Busy THEN
	iGroup.AddTrack(THIS^.fbTrack, THIS^.fbActiveCmd);
	AddToGroup := S_OK;
ELSE
	AddToGroup := S_FALSE;
END_IF
END_METHOD

METHOD RemoveFromGroup : HRESULT
IF NOT THIS^.fbActiveCmd.Busy THEN
	THIS^.fbTrack.RemoveFromGroup(THIS^.fbActiveCmd);
	RemoveFromGroup := S_OK;
ELSE
	RemoveFromGroup := S_FALSE;
END_IF
END_METHOD

METHOD AddMover : HRESULT
VAR_INPUT
	refMover : REFERENCE TO MC_PlanarMover;
	refFeedback : REFERENCE TO MC_PlanarFeedback;
END_VAR
refMover.JoinTrack(refFeedback, fbTrack, 0, 0);
END_METHOD

METHOD CalcTrackPoints : HRESULT
VAR_INPUT
END_VAR

VAR
    i         : UINT;
    oPosition : PositionXYC;
	fLength   : LREAL;
END_VAR
FOR i := 0 TO XplanarParameterlist.N_TRACE_POINTS DO
	fLength := THIS^.fbTrack.GetLength();
	THIS^.fbTrack.GetPositionAt(fLength/(XplanarParameterlist.N_TRACE_POINTS)*i, oPosition);
	
	THIS^.afTrackPoints[i].x := oPosition.x;
	THIS^.afTrackPoints[i].y := oPosition.y;
	THIS^.afTrackPoints[i].c := oPosition.c;
END_FOR

CalcTrackPoints := S_OK;
END_METHOD

METHOD Configure : HRESULT
VAR_INPUT
END_VAR
THIS^.nState_Configuring := 10;
Configure := S_OK;
END_METHOD

METHOD Abstract Configuring : HRESULT
END_METHOD

METHOD Disable : HRESULT
VAR_INPUT
END_VAR
IF NOT THIS^.fbActiveCmd.Busy THEN
	THIS^.fbTrack.Disable(fbActiveCmd);
	Disable := S_OK;
ELSE
	Disable := S_FALSE;
END_IF
END_METHOD

METHOD Enable : HRESULT
VAR_INPUT
END_VAR
IF NOT THIS^.fbActiveCmd.Busy THEN
	THIS^.fbTrack.Enable(fbActiveCmd);
	Enable := S_OK;
ELSE
	Enable := S_FALSE;
END_IF
END_METHOD

METHOD FB_init : BOOL
VAR_INPUT
	bInitRetains : BOOL; // if TRUE, the retain variables are initialized (warm start / cold start)
	bInCopyCode : BOOL;  // if TRUE, the instance afterwards gets moved into the copy code (online change)
	oSystem : I_CH_Object;
END_VAR
(* Register to the Xplanar System
   1. Test if the interface exists
   2. Test if the object implements a "System for Mover" interface 
*)
IF oSystem <> 0 AND_THEN __QUERYINTERFACE(oSystem,THIS^.iXpSystem) THEN
	THIS^.iXpSystem.RegisterTrack(THIS^);
END_IF
END_METHOD

{attribute 'monitoring':='call'}
PROPERTY HR : HRESULT
GET
IF THIS^.fbActiveCmd.Busy THEN
	HR := S_PENDING;
END_IF

IF THIS^.fbActiveCmd.Done THEN
	HR := S_OK;
END_IF

IF THIS^.fbActiveCmd.Error THEN
	HR := E_FAIL;
END_IF
END_GET
END_PROPERTY

{attribute 'monitoring':='call'}
PROPERTY Length : LREAL
GET
Length := THIS^.fbTrack.GetLength();
END_GET
END_PROPERTY

{attribute 'monitoring':='call'}
PROPERTY OID : OTCID
GET
OID := THIS^.fbTrack.MCTOPLC_STD.TrackOID;
END_GET
END_PROPERTY

{attribute 'monitoring':='call'}
PROPERTY PlanarTrack : REFERENCE TO MC_PlanarTrack
GET
PlanarTrack ref= THIS^.fbTrack;
END_GET
END_PROPERTY

METHOD Reset : HRESULT
VAR_INPUT
END_VAR
IF NOT THIS^.fbActiveCmd.Busy THEN
	THIS^.fbTrack.Reset(fbActiveCmd);
	Reset := S_OK;
ELSE
	Reset := S_FALSE;
END_IF
END_METHOD

METHOD PUBLIC Update : HRESULT
VAR_INPUT
END_VAR
THIS^.fbTrack.Update();
fbActiveCmd.Update();
END_METHOD

END_FUNCTION_BLOCK

// COMPONENTs/Track/FB_XP_Track_JSON
{attribute 'no_explicit_call' := '[FB_ImageSource] Do not call the body - Stick to OOP'}
FUNCTION_BLOCK FB_XP_Track_JSON EXTENDS FB_XP_Track_Base
VAR
	{attribute 'hide'}	
	fbJsonParser : FB_JsonDomParser;
END_VAR

METHOD ReadCenter : HRESULT;
VAR_INPUT
	oNode 	   : REFERENCE TO SJsonValue;
	fbCenter   : REFERENCE TO PositionXY;
END_VAR

VAR
	fX         : LREAL;
    fY         : LREAL;
	
	oProperty  : SJsonValue;
END_VAR
oProperty := fbJsonParser.FindMemberPath(oNode,'Center/X');
fX := fbJsonParser.GetDouble(oProperty);
oProperty := fbJsonParser.FindMemberPath(oNode,'Center/Y');
fY := fbJsonParser.GetDouble(oProperty);	
fbCenter.SetValuesXY(fX, fY);
END_METHOD

METHOD ReadDirection : HRESULT;
VAR_INPUT
	oNode 	   : REFERENCE TO SJsonValue;
	bClockwise : REFERENCE TO BOOL;
END_VAR

VAR
	oProperty  : SJsonValue;
END_VAR
oProperty := fbJsonParser.FindMemberPath(oNode,'Clockwise');
bClockwise := fbJsonParser.GetBool(oProperty);
END_METHOD

METHOD ReadEnd : HRESULT;
VAR_INPUT
	oNode 	   : REFERENCE TO SJsonValue;
	fbEnd	   : REFERENCE TO PositionXYC;
END_VAR

VAR
	fX         : LREAL;
    fY         : LREAL;
    fC         : LREAL;
	
	oProperty  : SJsonValue;
END_VAR
oProperty := THIS^.fbJsonParser.FindMemberPath(oNode,'End/X');
fX := fbJsonParser.GetDouble(oProperty);
oProperty := THIS^.fbJsonParser.FindMemberPath(oNode,'End/Y');
fY := fbJsonParser.GetDouble(oProperty);
oProperty := THIS^.fbJsonParser.FindMemberPath(oNode,'End/C');
fC := fbJsonParser.GetDouble(oProperty);
fbEnd.SetValuesXYC(fX, fY, fC);
END_METHOD

METHOD ReadStart : HRESULT;
VAR_INPUT
	oNode 	   : REFERENCE TO SJsonValue;
	fbStart	   : REFERENCE TO PositionXYC;
END_VAR

VAR
	fX         : LREAL;
    fY         : LREAL;
    fC         : LREAL;
	
	oProperty  : SJsonValue;
END_VAR
oProperty := THIS^.fbJsonParser.FindMemberPath(oNode,'Start/X');
fX := fbJsonParser.GetDouble(oProperty);
oProperty := THIS^.fbJsonParser.FindMemberPath(oNode,'Start/Y');
fY := fbJsonParser.GetDouble(oProperty);
oProperty := THIS^.fbJsonParser.FindMemberPath(oNode,'Start/C');
fC := fbJsonParser.GetDouble(oProperty);
fbStart.SetValuesXYC(fX, fY, fC);
END_METHOD

METHOD Configuring : HRESULT
VAR_INST
	iLinkedTrack : I_XP_Track;

    oDocument    : SJsonValue;
    bExec        : BOOL;
    sOID         : STRING(20);
    sPath        : STRING := XPlanarParameterlist.S_JSON_FOLDER_PATH_ON_TARGED;
    sPathFull    : STRING;
	
	oItr      : SJsonValue;
    oItrEnd   : SJsonValue;
END_VAR
VAR
    sType      : STRING(10);
    fX         : LREAL;
    fY         : LREAL;
    fC         : LREAL;
    fbStart    : PositionXYC;
    fbEnd      : PositionXYC;
    fbCenter   : PositionXY;
    bClockwise : BOOL;

    sLinkedOID   : STRING(20);
    oLinkedTrack : I_CH_Object;

    bClosed : BOOL;

    oOID      : SJsonValue;
    oSegments : SJsonValue;
    oProperty : SJsonValue;
END_VAR
Configuring := S_PENDING;
CASE nState_Configuring OF
	0: // Idle
		Configuring := S_OK;
		
	10:	// Configure file
		bExec := TRUE;
		sOID := DWORD_TO_HEXSTR(TO_DWORD(THIS^.OID),0,FALSE);
		sPathFull := CONCAT(sPath,sOID);
		sPathFull := CONCAT(sPathFull,'.JSON');	
		nState_Configuring := 20;
		
	20: // Load file
		fbJsonParser.LoadDocumentFromFile(sPathFull, bExec);
		IF NOT bExec THEN
			nState_Configuring := 30;
		END_IF
		
	30:	// Loading file		
		oDocument := fbJsonParser.GetDocumentRoot();
		nState_Configuring := 40;
	
	40: // Check file assgnment
		oOID := fbJsonParser.FindMember(oDocument, 'OID');
	  	IF (oOID <> 0) AND (fbJsonParser.GetString(oOID)=sOID) THEN
			nState_Configuring := 50;
		ELSE 
			nState_Configuring := 1000 + nState_Configuring;
	  	END_IF
		
	50: // Clear segments
		IF NOT THIS^.fbActiveCmd.Busy THEN
			THIS^.fbTrack.Clear(THIS^.fbActiveCmd);
			nState_Configuring := 52;
		END_IF
		
	52: // Clearing segments
		IF CheckOk(THIS^.HR) THEN 
			nState_Configuring := 61;
		ELSIF FAILED(THIS^.HR) THEN
			nState_Configuring := 1000 + nState_Configuring;
		END_IF	
		
	61: // Is an previous track defined?						
		IF fbJsonParser.HasMember(oDocument,'PreviousTrack') THEN
			oProperty := fbJsonParser.FindMember(oDocument,'PreviousTrack');
			sLinkedOID := fbJsonParser.GetString(oProperty);
			oLinkedTrack := THIS^.iXpSystem.Tracks.FindOIDString(sLinkedOID);
	
			IF ToTrack(oLinkedTrack,iLinkedTrack) THEN
				nState_Configuring := 62;
			ELSE
				nState_Configuring := 1000 + nState_Configuring;
			END_IF
		ELSE
			nState_Configuring := 70;
		END_IF
		
	62: // Link previous track 						
		// Wait for previous track to finish befor linking is posible 
		IF iLinkedTrack.Configuring() = S_OK THEN
			// Link previous track 
			THIS^.fbTrack.StartFromTrack(THIS^.fbActiveCmd, iLinkedTrack.PlanarTrack);
			nState_Configuring := 63;
		END_IF
	
	63: // Linking previous track 
		IF CheckOk(THIS^.HR) THEN 
			nState_Configuring := 70;
		ELSIF FAILED(THIS^.HR) THEN
			nState_Configuring := 1000 + nState_Configuring;
		END_IF	

	70:	// Load segment list
		oSegments := fbJsonParser.FindMember(oDocument, 'Segments');
		IF (oSegments <> 0) THEN		
		    oItr := fbJsonParser.ArrayBegin(oSegments);
		    oItrEnd := fbJsonParser.ArrayEnd(oSegments);
			
			nState_Configuring := 71;
		ELSE
			nState_Configuring := 1000 + nState_Configuring;
		END_IF	
			
	71: // Load single segment
		IF oItr <> 0 AND_THEN oItrEnd <> 0 AND_THEN oItr <> oItrEnd THEN
			(* Determine segment type *)
			oProperty := fbJsonParser.FindMember(oItr,'Type');
			sType := fbJsonParser.GetString(oProperty);
			
			(* For line types *)
			IF sType = 'Line' THEN
				THIS^.ReadStart(oNode := oItr, fbStart := fbStart);
				THIS^.ReadEnd(oNode := oItr, fbEnd := fbEnd);						
				THIS^.fbTrack.AppendLine(THIS^.fbActiveCmd, fbStart, fbEnd);
				
				nState_Configuring := 72;
				
			(* For circle types *)	
			ELSIF sType = 'Circle' THEN
				THIS^.ReadStart(oNode := oItr, fbStart := fbStart);
				THIS^.ReadEnd(oNode := oItr, fbEnd := fbEnd);
				THIS^.ReadCenter(oNode := oItr, fbCenter := fbCenter);
				THIS^.ReadDirection(oNode := oItr, bClockwise := bClockwise);
				THIS^.fbTrack.AppendCircle(THIS^.fbActiveCmd, fbStart, fbEnd, fbCenter, bClockwise);
				
				nState_Configuring := 72;
			ELSE
				//Not a valide sType	
				nState_Configuring := 1000 + nState_Configuring;
			END_IF
		ELSE
			nState_Configuring := 82;
		END_IF
			
	72: // Loading single segment - Loop
		IF CheckOk(THIS^.HR) THEN 
			oItr := fbJsonParser.NextArray(oItr);
			nState_Configuring := 71;
		ELSIF FAILED(THIS^.HR) THEN
			nState_Configuring := 1000 + nState_Configuring;
		END_IF		
		
	82: (* Link next track *)	
		IF fbJsonParser.HasMember(oDocument,'NextTrack') THEN
			oProperty := fbJsonParser.FindMember(oDocument,'NextTrack');
			sLinkedOID := fbJsonParser.GetString(oProperty);
			oLinkedTrack := THIS^.iXpSystem.Tracks.FindOIDString(sLinkedOID);
			
			IF ToTrack(oLinkedTrack,iLinkedTrack) THEN
				THIS^.fbTrack.EndAtTrack(THIS^.fbActiveCmd, iLinkedTrack.PlanarTrack);
				nState_Configuring := 83;
			END_IF
		ELSE
			nState_Configuring := 84;
		END_IF
		
	83: (* Linking next track *)	
		IF CheckOk(THIS^.HR) THEN 
			nState_Configuring := 84;
		ELSIF FAILED(THIS^.HR) THEN
			nState_Configuring := 1000 + nState_Configuring;
		END_IF

	84: (* Close the loop *)	
		IF fbJsonParser.HasMember(oDocument,'CloseLoop') THEN
			oProperty := fbJsonParser.FindMember(oDocument,'CloseLoop');
			bClosed := fbJsonParser.GetBool(oProperty);				
			IF bClosed THEN
				THIS^.fbTrack.CloseLoop(THIS^.fbActiveCmd);
				nState_Configuring := 85;
			ELSE
				nState_Configuring := 999;				
			END_IF
		ELSE
			nState_Configuring := 999;
		END_IF
		
	85: (* Closing the loop *)
		IF CheckOk(THIS^.HR) THEN 
			nState_Configuring := 999;
		ELSIF FAILED(THIS^.HR) THEN
			nState_Configuring := 1000 + nState_Configuring;
		END_IF
		
	999: // Done
		Configuring := S_OK;
		
	1000..1999://Error
		Configuring := E_FAIL;
END_CASE

IF fbJsonParser.ExceptionRaised() THEN
	nState_Configuring := 1000 + nState_Configuring;
	Configuring := E_FAIL;
END_IF
END_METHOD

END_FUNCTION_BLOCK

// COMPONENTs/Track/FB_XP_Track_TcCom
{attribute 'no_explicit_call' := '[FB_ImageSource] Do not call the body - Stick to OOP'}
FUNCTION_BLOCK FB_XP_Track_TcCom EXTENDS FB_XP_Track_Base
VAR

END_VAR

METHOD Configuring : HRESULT
Configuring := S_PENDING;
CASE nState_Configuring OF
	0: // Idle
		Configuring := S_OK;
		
	10: //Start
		//No config is done here. Set Track elements direkt in the Track TcCom Object
		nState_Configuring := 999;
		
	999: // Done
		Configuring := S_OK;
		
	1000..1999://Error
		Configuring := E_FAIL;
END_CASE
END_METHOD

END_FUNCTION_BLOCK
